LIN {X 0,Y 142.881,Z 390.405,A -85,B 0,C 180,E1 -25256.55,E2 -25256.55} C_VEL
LIN {X 0,Y 141.554,Z 401.416,A -85,B 0,C 180,E1 -25257.538,E2 -25257.538} C_VEL
LIN {X 0,Y 139.699,Z 412.081,A -85,B 0,C 180,E1 -25259.036,E2 -25259.036} C_VEL
LIN {X 0,Y 138.159,Z 420.57,A -85,B 0,C 180,E1 -25260.686,E2 -25260.686} C_VEL
LIN {X 0,Y 135.961,Z 428.897,A -85,B 0,C 180,E1 -25262.694,E2 -25262.694} C_VEL
LIN {X 0,Y 133.997,Z 436.865,A -85,B 0,C 180,E1 -25265.192,E2 -25265.192} C_VEL
LIN {X 0,Y 131.868,Z 444.276,A -85,B 0,C 180,E1 -25268.096,E2 -25268.096} C_VEL
LIN {X 0,Y 129.751,Z 451.798,A -85,B 0,C 180,E1 -25271.854,E2 -25271.854} C_VEL
LIN {X 0,Y 128.143,Z 457.67,A -85,B 0,C 180,E1 -25275.712,E2 -25275.712} C_VEL
LIN {X 0,Y 127.32,Z 461.5,A -85,B 0,C 180,E1 -25278.861,E2 -25278.861} C_VEL
LIN {X 0,Y 126.556,Z 465.852,A -85,B 0,C 180,E1 -25283.623,E2 -25283.623} C_VEL
LIN {X 0,Y 126.391,Z 468.069,A -85,B 0,C 180,E1 -25286.812,E2 -25286.812} C_VEL
LIN {X 0,Y 126.467,Z 469.672,A -85,B 0,C 180,E1 -25290,E2 -25290} C_VEL
LIN {X 0,Y 126.376,Z 470.674,A -85,B 0,C 180,E1 -25293.188,E2 -25293.188} C_VEL
LIN {X 0,Y 126.521,Z 471.21,A -85,B 0,C 180,E1 -25296.378,E2 -25296.378} C_VEL
LIN {X 0,Y 126.968,Z 471.301,A -85,B 0,C 180,E1 -25299.558,E2 -25299.558} C_VEL
LIN {X 0,Y 127.775,Z 470.915,A -85,B 0,C 180,E1 -25302.709,E2 -25302.709} C_VEL
LIN {X 0,Y 128.973,Z 469.949,A -85,B 0,C 180,E1 -25305.81,E2 -25305.81} C_VEL
LIN {X 0,Y 130.517,Z 468.51,A -85,B 0,C 180,E1 -25308.849,E2 -25308.849} C_VEL
LIN {X 0,Y 133.483,Z 465.427,A -85,B 0,C 180,E1 -25313.258,E2 -25313.258} C_VEL
LIN {X 0,Y 137.366,Z 461.085,A -85,B 0,C 180,E1 -25317.416,E2 -25317.416} C_VEL
LIN {X 0,Y 141.882,Z 455.129,A -85,B 0,C 180,E1 -25321.338,E2 -25321.338} C_VEL
LIN {X 0,Y 146.264,Z 448.82,A -85,B 0,C 180,E1 -25324.372,E2 -25324.372} C_VEL
LIN {X 0,Y 149.954,Z 442.696,A -85,B 0,C 180,E1 -25326.694,E2 -25326.694} C_VEL
LIN {X 0,Y 153.372,Z 436.478,A -85,B 0,C 180,E1 -25328.55,E2 -25328.55} C_VEL
LIN {X 0,Y 156.553,Z 429.785,A -85,B 0,C 180,E1 -25330.188,E2 -25330.188} C_VEL
LIN {X 0,Y 159.841,Z 421.95,A -85,B 0,C 180,E1 -25331.683,E2 -25331.683} C_VEL
LIN {X 0,Y 162.735,Z 413.909,A -85,B 0,C 180,E1 -25332.857,E2 -25332.857} C_VEL
LIN {X 0,Y 165.005,Z 406.242,A -85,B 0,C 180,E1 -25333.73,E2 -25333.73} C_VEL
LIN {X 0,Y 165.605,Z 401.983,A -85,B 0,C 180,E1 -25334.367,E2 -25334.367} C_VEL
LIN {X 0,Y 164.474,Z 391.08,A -85,B 0,C 180,E1 -25336.71,E2 -25336.71} C_VEL
LIN {X 0,Y 164.587,Z 387.258,A -85,B 0,C 180,E1 -25337.085,E2 -25337.085} C_VEL
LIN {X 0,Y 165.584,Z 377.046,A -85,B 0,C 180,E1 -25337.548,E2 -25337.548} C_VEL
LIN {X 0,Y 163.149,Z 370.127,A -85,B 0,C 180,E1 -25339.553,E2 -25339.553} C_VEL
LIN {X 0,Y 160.189,Z 363.188,A -85,B 0,C 180,E1 -25342.105,E2 -25342.105} C_VEL
LIN {X 0,Y 157.036,Z 356.535,A -85,B 0,C 180,E1 -25345.217,E2 -25345.217} C_VEL
LIN {X 0,Y 155.41,Z 353.618,A -85,B 0,C 180,E1 -25346.981,E2 -25346.981} C_VEL
LIN {X 0,Y 152.992,Z 349.888,A -85,B 0,C 180,E1 -25349.954,E2 -25349.954} C_VEL
LIN {X 0,Y 150.142,Z 345.841,A -85,B 0,C 180,E1 -25354.422,E2 -25354.422} C_VEL
LIN {X 0,Y 149.876,Z 345.124,A -85,B 0,C 180,E1 -25355.038,E2 -25355.038} C_VEL
LIN {X 0,Y 147.126,Z 341.865,A -85,B 0,C 180,E1 -25364.768,E2 -25364.768} C_VEL
LIN {X 0,Y 147.088,Z 341.6,A -85,B 0,C 180,E1 -25366.178,E2 -25366.178} C_VEL
LIN {X 0,Y 147.398,Z 341.979,A -85,B 0,C 180,E1 -25369.849,E2 -25369.849} C_VEL
LIN {X 0,Y 149.892,Z 344.586,A -85,B 0,C 180,E1 -25377.313,E2 -25377.313} C_VEL
LIN {X 0,Y 150.355,Z 345.232,A -85,B 0,C 180,E1 -25378.236,E2 -25378.236} C_VEL
LIN {X 0,Y 152.17,Z 348.533,A -85,B 0,C 180,E1 -25381.324,E2 -25381.324} C_VEL
LIN {X 0,Y 153.507,Z 350.114,A -85,B 0,C 180,E1 -25383.105,E2 -25383.105} C_VEL
LIN {X 0,Y 156.121,Z 354.377,A -85,B 0,C 180,E1 -25386.209,E2 -25386.209} C_VEL
LIN {X 0,Y 159.1,Z 359.359,A -85,B 0,C 180,E1 -25389.17,E2 -25389.17} C_VEL
LIN {X 0,Y 162.048,Z 364.517,A -85,B 0,C 180,E1 -25391.701,E2 -25391.701} C_VEL
LIN {X 0,Y 165.657,Z 371.579,A -85,B 0,C 180,E1 -25394.47,E2 -25394.47} C_VEL
LIN {X 0,Y 165.925,Z 372.264,A -85,B 0,C 180,E1 -25394.677,E2 -25394.677} C_VEL
LIN {X 0,Y 164.165,Z 387.712,A -85,B 0,C 180,E1 -25395.387,E2 -25395.387} C_VEL
LIN {X 0,Y 162.262,Z 397.3,A -85,B 0,C 180,E1 -25396.153,E2 -25396.153} C_VEL
LIN {X 0,Y 159.595,Z 407.073,A -85,B 0,C 180,E1 -25397.253,E2 -25397.253} C_VEL
LIN {X 0,Y 156.834,Z 415.193,A -85,B 0,C 180,E1 -25398.467,E2 -25398.467} C_VEL
LIN {X 0,Y 153.338,Z 423.473,A -85,B 0,C 180,E1 -25400.023,E2 -25400.023} C_VEL
LIN {X 0,Y 149.693,Z 430.879,A -85,B 0,C 180,E1 -25401.83,E2 -25401.83} C_VEL
LIN {X 0,Y 145.991,Z 437.405,A -85,B 0,C 180,E1 -25403.847,E2 -25403.847} C_VEL
LIN {X 0,Y 141.45,Z 444.337,A -85,B 0,C 180,E1 -25406.581,E2 -25406.581} C_VEL
LIN {X 0,Y 137.261,Z 449.948,A -85,B 0,C 180,E1 -25409.495,E2 -25409.495} C_VEL
LIN {X 0,Y 133.417,Z 454.459,A -85,B 0,C 180,E1 -25412.563,E2 -25412.563} C_VEL
LIN {X 0,Y 129.233,Z 458.881,A -85,B 0,C 180,E1 -25416.742,E2 -25416.742} C_VEL
LIN {X 0,Y 127.087,Z 460.797,A -85,B 0,C 180,E1 -25419.269,E2 -25419.269} C_VEL
LIN {X 0,Y 124.55,Z 462.795,A -85,B 0,C 180,E1 -25422.817,E2 -25422.817} C_VEL
LIN {X 0,Y 121.52,Z 464.62,A -85,B 0,C 180,E1 -25428.751,E2 -25428.751} C_VEL
LIN {X 0,Y 119.539,Z 464.603,A -85,B 0,C 180,E1 -25435.397,E2 -25435.397} C_VEL
LIN {X 0,Y 119.135,Z 464.109,A -85,B 0,C 180,E1 -25437.933,E2 -25437.933} C_VEL
LIN {X 0,Y 118.875,Z 462.498,A -85,B 0,C 180,E1 -25442.476,E2 -25442.476} C_VEL
LIN {X 0,Y 119.08,Z 460.912,A -85,B 0,C 180,E1 -25445.599,E2 -25445.599} C_VEL
LIN {X 0,Y 119.74,Z 457.829,A -85,B 0,C 180,E1 -25449.903,E2 -25449.903} C_VEL
LIN {X 0,Y 121.008,Z 452.9,A -85,B 0,C 180,E1 -25454.85,E2 -25454.85} C_VEL
LIN {X 0,Y 122.587,Z 447.322,A -85,B 0,C 180,E1 -25459.097,E2 -25459.097} C_VEL
LIN {X 0,Y 124.429,Z 441.266,A -85,B 0,C 180,E1 -25462.699,E2 -25462.699} C_VEL
LIN {X 0,Y 126.768,Z 433.558,A -85,B 0,C 180,E1 -25466.309,E2 -25466.309} C_VEL
LIN {X 0,Y 129.417,Z 424.126,A -85,B 0,C 180,E1 -25469.611,E2 -25469.611} C_VEL
LIN {X 0,Y 131.533,Z 415.611,A -85,B 0,C 180,E1 -25471.914,E2 -25471.914} C_VEL
LIN {X 0,Y 133.45,Z 406.731,A -85,B 0,C 180,E1 -25473.773,E2 -25473.773} C_VEL
LIN {X 0,Y 134.912,Z 397.798,A -85,B 0,C 180,E1 -25475.218,E2 -25475.218} C_VEL
LIN {X 0,Y 136.377,Z 386.472,A -85,B 0,C 180,E1 -25476.512,E2 -25476.512} C_VEL
LIN {X 0,Y 137.535,Z 371.795,A -85,B 0,C 180,E1 -25477.412,E2 -25477.412} C_VEL
LIN {X 0,Y 138.736,Z 349.669,A -85,B 0,C 180,E1 -25478.553,E2 -25478.553} C_VEL
LIN {X 0,Y 136.797,Z 343.639,A -85,B 0,C 180,E1 -25479.381,E2 -25479.381} C_VEL
LIN {X 0,Y 128.682,Z 327.088,A -85,B 0,C 180,E1 -25482.589,E2 -25482.589} C_VEL
LIN {X 0,Y 123.725,Z 318.724,A -85,B 0,C 180,E1 -25484.659,E2 -25484.659} C_VEL
LIN {X 0,Y 122.333,Z 316.065,A -85,B 0,C 180,E1 -25485.299,E2 -25485.299} C_VEL
LIN {X 0,Y 122.147,Z 315.082,A -85,B 0,C 180,E1 -25485.541,E2 -25485.541} C_VEL
LIN {X 0,Y 122.023,Z 315.065,A -85,B 0,C 180,E1 -25492.848,E2 -25492.848} C_VEL
LIN {X 0,Y 121.957,Z 315.112,A -85,B 0,C 180,E1 -25497.452,E2 -25497.452} C_VEL
LIN {X 0,Y 121.904,Z 315.107,A -85,B 0,C 180,E1 -25501.255,E2 -25501.255} C_VEL
LIN {X 0,Y 121.886,Z 315.116,A -85,B 0,C 180,E1 -25506.171,E2 -25506.171} C_VEL
LIN {X 0,Y 121.88,Z 315.098,A -85,B 0,C 180,E1 -25511.442,E2 -25511.442} C_VEL
LIN {X 0,Y 121.925,Z 315.109,A -85,B 0,C 180,E1 -25518.532,E2 -25518.532} C_VEL
LIN {X 0,Y 121.95,Z 315.077,A -85,B 0,C 180,E1 -25524.809,E2 -25524.809} C_VEL
LIN {X 0,Y 121.927,Z 315.105,A -85,B 0,C 180,E1 -25529.836,E2 -25529.836} C_VEL
LIN {X 0,Y 121.98,Z 315.086,A -85,B 0,C 180,E1 -25536.214,E2 -25536.214} C_VEL
LIN {X 0,Y 122.04,Z 315.06,A -85,B 0,C 180,E1 -25539.786,E2 -25539.786} C_VEL
LIN {X 0,Y 122.236,Z 315.072,A -85,B 0,C 180,E1 -25546.704,E2 -25546.704} C_VEL
LIN {X 0,Y 122.403,Z 315.044,A -85,B 0,C 180,E1 -25550.081,E2 -25550.081} C_VEL
LIN {X 0,Y 122.589,Z 315,A -85,B 0,C 180,E1 -25556.713,E2 -25556.713} C_VEL
LIN {X 0,Y 123.036,Z 314.966,A -85,B 0,C 180,E1 -25560,E2 -25560} C_VEL
LIN {X 0,Y 122.419,Z 315.034,A -85,B 0,C 180,E1 -25566.593,E2 -25566.593} C_VEL
LIN {X 0,Y 122.319,Z 315.049,A -85,B 0,C 180,E1 -25572.385,E2 -25572.385} C_VEL
LIN {X 0,Y 122.1,Z 315.087,A -85,B 0,C 180,E1 -25576.726,E2 -25576.726} C_VEL
LIN {X 0,Y 122.024,Z 315.084,A -85,B 0,C 180,E1 -25582.855,E2 -25582.855} C_VEL
LIN {X 0,Y 121.937,Z 315.108,A -85,B 0,C 180,E1 -25587.457,E2 -25587.457} C_VEL
LIN {X 0,Y 121.896,Z 315.103,A -85,B 0,C 180,E1 -25591.258,E2 -25591.258} C_VEL
LIN {X 0,Y 121.88,Z 315.114,A -85,B 0,C 180,E1 -25596.171,E2 -25596.171} C_VEL
LIN {X 0,Y 121.861,Z 315.085,A -85,B 0,C 180,E1 -25601.434,E2 -25601.434} C_VEL
LIN {X 0,Y 121.869,Z 315.22,A -85,B 0,C 180,E1 -25606.089,E2 -25606.089} C_VEL
LIN {X 0,Y 122.984,Z 318.162,A -85,B 0,C 180,E1 -25606.67,E2 -25606.67} C_VEL
LIN {X 0,Y 124.377,Z 320.409,A -85,B 0,C 180,E1 -25607.271,E2 -25607.271} C_VEL
LIN {X 0,Y 129.513,Z 329.802,A -85,B 0,C 180,E1 -25609.438,E2 -25609.438} C_VEL
LIN {X 0,Y 134.184,Z 342.151,A -85,B 0,C 180,E1 -25611.496,E2 -25611.496} C_VEL
LIN {X 0,Y 136.431,Z 349.354,A -85,B 0,C 180,E1 -25612.502,E2 -25612.502} C_VEL
LIN {X 0,Y 137.956,Z 367.641,A -85,B 0,C 180,E1 -25614.015,E2 -25614.015} C_VEL
LIN {X 0,Y 136.489,Z 390.702,A -85,B 0,C 180,E1 -25615.297,E2 -25615.297} C_VEL
LIN {X 0,Y 135.015,Z 402.002,A -85,B 0,C 180,E1 -25616.379,E2 -25616.379} C_VEL
LIN {X 0,Y 133.188,Z 411.946,A -85,B 0,C 180,E1 -25617.848,E2 -25617.848} C_VEL
LIN {X 0,Y 131.625,Z 420.222,A -85,B 0,C 180,E1 -25619.521,E2 -25619.521} C_VEL
LIN {X 0,Y 129.328,Z 428.565,A -85,B 0,C 180,E1 -25621.609,E2 -25621.609} C_VEL
LIN {X 0,Y 127.262,Z 436.553,A -85,B 0,C 180,E1 -25624.222,E2 -25624.222} C_VEL
LIN {X 0,Y 125.304,Z 443.124,A -85,B 0,C 180,E1 -25626.883,E2 -25626.883} C_VEL
LIN {X 0,Y 123.38,Z 449.369,A -85,B 0,C 180,E1 -25630.016,E2 -25630.016} C_VEL
LIN {X 0,Y 121.893,Z 454.554,A -85,B 0,C 180,E1 -25633.245,E2 -25633.245} C_VEL
LIN {X 0,Y 120.763,Z 458.86,A -85,B 0,C 180,E1 -25636.539,E2 -25636.539} C_VEL
LIN {X 0,Y 119.968,Z 462.417,A -85,B 0,C 180,E1 -25639.878,E2 -25639.878} C_VEL
LIN {X 0,Y 119.386,Z 466.474,A -85,B 0,C 180,E1 -25644.934,E2 -25644.934} C_VEL
LIN {X 0,Y 119.315,Z 467.602,A -85,B 0,C 180,E1 -25646.623,E2 -25646.623} C_VEL
LIN {X 0,Y 119.39,Z 469.238,A -85,B 0,C 180,E1 -25650,E2 -25650} C_VEL
LIN {X 0,Y 119.285,Z 470.332,A -85,B 0,C 180,E1 -25653.378,E2 -25653.378} C_VEL
LIN {X 0,Y 119.462,Z 470.963,A -85,B 0,C 180,E1 -25656.757,E2 -25656.757} C_VEL
LIN {X 0,Y 119.972,Z 471.15,A -85,B 0,C 180,E1 -25660.121,E2 -25660.121} C_VEL
LIN {X 0,Y 120.85,Z 470.781,A -85,B 0,C 180,E1 -25663.451,E2 -25663.451} C_VEL
LIN {X 0,Y 122.135,Z 469.894,A -85,B 0,C 180,E1 -25666.721,E2 -25666.721} C_VEL
LIN {X 0,Y 123.811,Z 468.554,A -85,B 0,C 180,E1 -25669.912,E2 -25669.912} C_VEL
LIN {X 0,Y 127,Z 465.575,A -85,B 0,C 180,E1 -25674.521,E2 -25674.521} C_VEL
LIN {X 0,Y 129.642,Z 462.894,A -85,B 0,C 180,E1 -25677.437,E2 -25677.437} C_VEL
LIN {X 0,Y 134.245,Z 457.71,A -85,B 0,C 180,E1 -25681.567,E2 -25681.567} C_VEL
LIN {X 0,Y 138.626,Z 452.168,A -85,B 0,C 180,E1 -25684.773,E2 -25684.773} C_VEL
LIN {X 0,Y 143.403,Z 445.255,A -85,B 0,C 180,E1 -25687.777,E2 -25687.777} C_VEL
LIN {X 0,Y 147.966,Z 437.517,A -85,B 0,C 180,E1 -25690.27,E2 -25690.27} C_VEL
LIN {X 0,Y 152.028,Z 429.463,A -85,B 0,C 180,E1 -25692.268,E2 -25692.268} C_VEL
LIN {X 0,Y 155.268,Z 422.18,A -85,B 0,C 180,E1 -25693.65,E2 -25693.65} C_VEL
LIN {X 0,Y 158.274,Z 414.242,A -85,B 0,C 180,E1 -25694.821,E2 -25694.821} C_VEL
LIN {X 0,Y 160.984,Z 405.406,A -85,B 0,C 180,E1 -25695.812,E2 -25695.812} C_VEL
LIN {X 0,Y 163.083,Z 396.249,A -85,B 0,C 180,E1 -25696.588,E2 -25696.588} C_VEL
LIN {X 0,Y 164.587,Z 387.258,A -85,B 0,C 180,E1 -25697.085,E2 -25697.085} C_VEL
LIN {X 0,Y 164.625,Z 384.216,A -85,B 0,C 180,E1 -25697.418,E2 -25697.418} C_VEL
LIN {X 0,Y 163.648,Z 380.573,A -85,B 0,C 180,E1 -25698.321,E2 -25698.321} C_VEL
LIN {X 0,Y 162.806,Z 378.841,A -85,B 0,C 180,E1 -25698.965,E2 -25698.965} C_VEL
LIN {X 0,Y 158.938,Z 372.15,A -85,B 0,C 180,E1 -25702.014,E2 -25702.014} C_VEL
LIN {X 0,Y 156.045,Z 365.237,A -85,B 0,C 180,E1 -25704.964,E2 -25704.964} C_VEL
LIN {X 0,Y 153.632,Z 360.182,A -85,B 0,C 180,E1 -25707.728,E2 -25707.728} C_VEL
LIN {X 0,Y 151.299,Z 356.419,A -85,B 0,C 180,E1 -25710.824,E2 -25710.824} C_VEL
LIN {X 0,Y 148.68,Z 352.346,A -85,B 0,C 180,E1 -25715.359,E2 -25715.359} C_VEL
LIN {X 0,Y 148.117,Z 351.687,A -85,B 0,C 180,E1 -25716.594,E2 -25716.594} C_VEL
LIN {X 0,Y 146.134,Z 348.78,A -85,B 0,C 180,E1 -25725.376,E2 -25725.376} C_VEL
LIN {X 0,Y 146.36,Z 348.904,A -85,B 0,C 180,E1 -25729.355,E2 -25729.355} C_VEL
LIN {X 0,Y 148.716,Z 351.517,A -85,B 0,C 180,E1 -25736.953,E2 -25736.953} C_VEL
LIN {X 0,Y 150.98,Z 355.613,A -85,B 0,C 180,E1 -25741.112,E2 -25741.112} C_VEL
LIN {X 0,Y 151.99,Z 357.05,A -85,B 0,C 180,E1 -25742.54,E2 -25742.54} C_VEL
LIN {X 0,Y 154.147,Z 360.784,A -85,B 0,C 180,E1 -25745.304,E2 -25745.304} C_VEL
LIN {X 0,Y 157.613,Z 366.789,A -85,B 0,C 180,E1 -25748.904,E2 -25748.904} C_VEL
LIN {X 0,Y 161.88,Z 375.319,A -85,B 0,C 180,E1 -25752.643,E2 -25752.643} C_VEL
LIN {X 0,Y 160.367,Z 387.956,A -85,B 0,C 180,E1 -25753.275,E2 -25753.275} C_VEL
LIN {X 0,Y 158.275,Z 397.956,A -85,B 0,C 180,E1 -25754.078,E2 -25754.078} C_VEL
LIN {X 0,Y 155.458,Z 407.697,A -85,B 0,C 180,E1 -25755.17,E2 -25755.17} C_VEL
LIN {X 0,Y 152.131,Z 416.773,A -85,B 0,C 180,E1 -25756.553,E2 -25756.553} C_VEL
LIN {X 0,Y 148.716,Z 424.307,A -85,B 0,C 180,E1 -25758.005,E2 -25758.005} C_VEL
LIN {X 0,Y 144.809,Z 431.748,A -85,B 0,C 180,E1 -25759.861,E2 -25759.861} C_VEL
LIN {X 0,Y 140.404,Z 438.966,A -85,B 0,C 180,E1 -25762.181,E2 -25762.181} C_VEL
LIN {X 0,Y 134.426,Z 447.162,A -85,B 0,C 180,E1 -25765.739,E2 -25765.739} C_VEL
LIN {X 0,Y 131.257,Z 451.035,A -85,B 0,C 180,E1 -25767.943,E2 -25767.943} C_VEL
LIN {X 0,Y 127.214,Z 455.365,A -85,B 0,C 180,E1 -25771.099,E2 -25771.099} C_VEL
LIN {X 0,Y 123.456,Z 458.98,A -85,B 0,C 180,E1 -25774.7,E2 -25774.7} C_VEL
LIN {X 0,Y 120.51,Z 461.436,A -85,B 0,C 180,E1 -25778.068,E2 -25778.068} C_VEL
LIN {X 0,Y 116.677,Z 463.957,A -85,B 0,C 180,E1 -25783.714,E2 -25783.714} C_VEL
LIN {X 0,Y 114.749,Z 464.846,A -85,B 0,C 180,E1 -25787.647,E2 -25787.647} C_VEL
LIN {X 0,Y 113.333,Z 465.087,A -85,B 0,C 180,E1 -25791.677,E2 -25791.677} C_VEL
LIN {X 0,Y 112.367,Z 464.659,A -85,B 0,C 180,E1 -25795.744,E2 -25795.744} C_VEL
LIN {X 0,Y 111.773,Z 462.831,A -85,B 0,C 180,E1 -25801.677,E2 -25801.677} C_VEL
LIN {X 0,Y 112.31,Z 459.382,A -85,B 0,C 180,E1 -25807.948,E2 -25807.948} C_VEL
LIN {X 0,Y 113.072,Z 456.268,A -85,B 0,C 180,E1 -25811.895,E2 -25811.895} C_VEL
LIN {X 0,Y 114.125,Z 452.411,A -85,B 0,C 180,E1 -25815.74,E2 -25815.74} C_VEL
LIN {X 0,Y 115.945,Z 446.423,A -85,B 0,C 180,E1 -25820.405,E2 -25820.405} C_VEL
LIN {X 0,Y 118.369,Z 438.758,A -85,B 0,C 180,E1 -25824.891,E2 -25824.891} C_VEL
LIN {X 0,Y 120.764,Z 430.977,A -85,B 0,C 180,E1 -25828.333,E2 -25828.333} C_VEL
LIN {X 0,Y 122.829,Z 423.921,A -85,B 0,C 180,E1 -25830.82,E2 -25830.82} C_VEL
LIN {X 0,Y 125.081,Z 415.306,A -85,B 0,C 180,E1 -25833.221,E2 -25833.221} C_VEL
LIN {X 0,Y 127.001,Z 406.766,A -85,B 0,C 180,E1 -25835.065,E2 -25835.065} C_VEL
LIN {X 0,Y 128.531,Z 397.81,A -85,B 0,C 180,E1 -25836.565,E2 -25836.565} C_VEL
LIN {X 0,Y 130.127,Z 385.909,A -85,B 0,C 180,E1 -25837.948,E2 -25837.948} C_VEL
LIN {X 0,Y 131.444,Z 369.026,A -85,B 0,C 180,E1 -25838.966,E2 -25838.966} C_VEL
LIN {X 0,Y 132.421,Z 350.923,A -85,B 0,C 180,E1 -25839.948,E2 -25839.948} C_VEL
LIN {X 0,Y 131.134,Z 347.005,A -85,B 0,C 180,E1 -25840.537,E2 -25840.537} C_VEL
LIN {X 0,Y 123.12,Z 330.389,A -85,B 0,C 180,E1 -25843.974,E2 -25843.974} C_VEL
LIN {X 0,Y 116.777,Z 319.818,A -85,B 0,C 180,E1 -25846.876,E2 -25846.876} C_VEL
LIN {X 0,Y 115.222,Z 317.086,A -85,B 0,C 180,E1 -25847.666,E2 -25847.666} C_VEL
LIN {X 0,Y 114.975,Z 315.967,A -85,B 0,C 180,E1 -25847.911,E2 -25847.911} C_VEL
LIN {X 0,Y 114.946,Z 315.95,A -85,B 0,C 180,E1 -25853.49,E2 -25853.49} C_VEL
LIN {X 0,Y 114.862,Z 315.984,A -85,B 0,C 180,E1 -25861.061,E2 -25861.061} C_VEL
LIN {X 0,Y 114.782,Z 316.001,A -85,B 0,C 180,E1 -25867.754,E2 -25867.754} C_VEL
LIN {X 0,Y 114.807,Z 315.975,A -85,B 0,C 180,E1 -25872.727,E2 -25872.727} C_VEL
LIN {X 0,Y 114.844,Z 315.992,A -85,B 0,C 180,E1 -25877.688,E2 -25877.688} C_VEL
LIN {X 0,Y 114.847,Z 315.971,A -85,B 0,C 180,E1 -25882.703,E2 -25882.703} C_VEL
LIN {X 0,Y 114.862,Z 315.983,A -85,B 0,C 180,E1 -25888.935,E2 -25888.935} C_VEL
LIN {X 0,Y 114.945,Z 315.96,A -85,B 0,C 180,E1 -25896.507,E2 -25896.507} C_VEL
LIN {X 0,Y 115.007,Z 315.953,A -85,B 0,C 180,E1 -25902.209,E2 -25902.209} C_VEL
LIN {X 0,Y 115.252,Z 315.941,A -85,B 0,C 180,E1 -25907.327,E2 -25907.327} C_VEL
LIN {X 0,Y 115.359,Z 315.901,A -85,B 0,C 180,E1 -25913.001,E2 -25913.001} C_VEL
LIN {X 0,Y 115.988,Z 315.844,A -85,B 0,C 180,E1 -25920,E2 -25920} C_VEL
LIN {X 0,Y 115.36,Z 315.909,A -85,B 0,C 180,E1 -25926.998,E2 -25926.998} C_VEL
LIN {X 0,Y 115.252,Z 315.931,A -85,B 0,C 180,E1 -25932.671,E2 -25932.671} C_VEL
LIN {X 0,Y 115.004,Z 315.967,A -85,B 0,C 180,E1 -25937.791,E2 -25937.791} C_VEL
LIN {X 0,Y 114.944,Z 315.97,A -85,B 0,C 180,E1 -25943.492,E2 -25943.492} C_VEL
LIN {X 0,Y 114.853,Z 315.979,A -85,B 0,C 180,E1 -25951.057,E2 -25951.057} C_VEL
LIN {X 0,Y 114.774,Z 315.986,A -85,B 0,C 180,E1 -25957.758,E2 -25957.758} C_VEL
LIN {X 0,Y 114.784,Z 315.984,A -85,B 0,C 180,E1 -25963.678,E2 -25963.678} C_VEL
LIN {X 0,Y 115.813,Z 318.882,A -85,B 0,C 180,E1 -25964.3,E2 -25964.3} C_VEL
LIN {X 0,Y 117.212,Z 320.888,A -85,B 0,C 180,E1 -25964.962,E2 -25964.962} C_VEL
LIN {X 0,Y 123.967,Z 333.026,A -85,B 0,C 180,E1 -25968.08,E2 -25968.08} C_VEL
LIN {X 0,Y 128.513,Z 345.387,A -85,B 0,C 180,E1 -25970.267,E2 -25970.267} C_VEL
LIN {X 0,Y 130.313,Z 351.13,A -85,B 0,C 180,E1 -25971.138,E2 -25971.138} C_VEL
LIN {X 0,Y 131.654,Z 368.464,A -85,B 0,C 180,E1 -25972.646,E2 -25972.646} C_VEL
LIN {X 0,Y 130.172,Z 390.427,A -85,B 0,C 180,E1 -25973.916,E2 -25973.916} C_VEL
LIN {X 0,Y 128.515,Z 402.447,A -85,B 0,C 180,E1 -25975.131,E2 -25975.131} C_VEL
LIN {X 0,Y 126.537,Z 412.644,A -85,B 0,C 180,E1 -25976.739,E2 -25976.739} C_VEL
LIN {X 0,Y 124.736,Z 421.206,A -85,B 0,C 180,E1 -25978.59,E2 -25978.59} C_VEL
LIN {X 0,Y 122.381,Z 429.343,A -85,B 0,C 180,E1 -25980.783,E2 -25980.783} C_VEL
LIN {X 0,Y 120.568,Z 436.148,A -85,B 0,C 180,E1 -25983.145,E2 -25983.145} C_VEL
LIN {X 0,Y 118.219,Z 443.608,A -85,B 0,C 180,E1 -25986.342,E2 -25986.342} C_VEL
LIN {X 0,Y 115.874,Z 451.178,A -85,B 0,C 180,E1 -25990.514,E2 -25990.514} C_VEL
LIN {X 0,Y 113.861,Z 458.084,A -85,B 0,C 180,E1 -25995.706,E2 -25995.706} C_VEL
LIN {X 0,Y 112.682,Z 463.288,A -85,B 0,C 180,E1 -26001.03,E2 -26001.03} C_VEL
LIN {X 0,Y 112.245,Z 467.079,A -85,B 0,C 180,E1 -26006.41,E2 -26006.41} C_VEL
LIN {X 0,Y 112.301,Z 468.797,A -85,B 0,C 180,E1 -26010,E2 -26010} C_VEL
LIN {X 0,Y 112.204,Z 469.989,A -85,B 0,C 180,E1 -26013.591,E2 -26013.591} C_VEL
LIN {X 0,Y 112.425,Z 470.718,A -85,B 0,C 180,E1 -26017.182,E2 -26017.182} C_VEL
LIN {X 0,Y 112.973,Z 470.964,A -85,B 0,C 180,E1 -26020.756,E2 -26020.756} C_VEL
LIN {X 0,Y 113.955,Z 470.632,A -85,B 0,C 180,E1 -26024.281,E2 -26024.281} C_VEL
LIN {X 0,Y 115.335,Z 469.846,A -85,B 0,C 180,E1 -26027.738,E2 -26027.738} C_VEL
LIN {X 0,Y 117.137,Z 468.613,A -85,B 0,C 180,E1 -26031.099,E2 -26031.099} C_VEL
LIN {X 0,Y 119.277,Z 466.907,A -85,B 0,C 180,E1 -26034.358,E2 -26034.358} C_VEL
LIN {X 0,Y 123.4,Z 463.19,A -85,B 0,C 180,E1 -26038.952,E2 -26038.952} C_VEL
LIN {X 0,Y 126.608,Z 460.041,A -85,B 0,C 180,E1 -26041.825,E2 -26041.825} C_VEL
LIN {X 0,Y 130.964,Z 455.07,A -85,B 0,C 180,E1 -26045.23,E2 -26045.23} C_VEL
LIN {X 0,Y 135.807,Z 448.852,A -85,B 0,C 180,E1 -26048.388,E2 -26048.388} C_VEL
LIN {X 0,Y 139.922,Z 442.814,A -85,B 0,C 180,E1 -26050.764,E2 -26050.764} C_VEL
LIN {X 0,Y 144.471,Z 435.495,A -85,B 0,C 180,E1 -26052.924,E2 -26052.924} C_VEL
LIN {X 0,Y 148.499,Z 427.674,A -85,B 0,C 180,E1 -26054.773,E2 -26054.773} C_VEL
LIN {X 0,Y 152.778,Z 418.092,A -85,B 0,C 180,E1 -26056.427,E2 -26056.427} C_VEL
LIN {X 0,Y 156.539,Z 407.168,A -85,B 0,C 180,E1 -26057.775,E2 -26057.775} C_VEL
LIN {X 0,Y 159.103,Z 396.879,A -85,B 0,C 180,E1 -26058.669,E2 -26058.669} C_VEL
LIN {X 0,Y 160.801,Z 387.378,A -85,B 0,C 180,E1 -26059.194,E2 -26059.194} C_VEL
LIN {X 0,Y 161.595,Z 379.591,A -85,B 0,C 180,E1 -26059.586,E2 -26059.586} C_VEL
LIN {X 0,Y 158.938,Z 372.15,A -85,B 0,C 180,E1 -26062.014,E2 -26062.014} C_VEL
LIN {X 0,Y 157.126,Z 368.923,A -85,B 0,C 180,E1 -26063.678,E2 -26063.678} C_VEL
LIN {X 0,Y 155.073,Z 366.798,A -85,B 0,C 180,E1 -26065.573,E2 -26065.573} C_VEL
LIN {X 0,Y 149.985,Z 363.317,A -85,B 0,C 180,E1 -26071.22,E2 -26071.22} C_VEL
LIN {X 0,Y 149.019,Z 362.194,A -85,B 0,C 180,E1 -26072.677,E2 -26072.677} C_VEL
LIN {X 0,Y 147.203,Z 358.783,A -85,B 0,C 180,E1 -26076.44,E2 -26076.44} C_VEL
LIN {X 0,Y 145.162,Z 355.8,A -85,B 0,C 180,E1 -26085.527,E2 -26085.527} C_VEL
LIN {X 0,Y 145.378,Z 355.962,A -85,B 0,C 180,E1 -26089.282,E2 -26089.282} C_VEL
LIN {X 0,Y 147.565,Z 358.67,A -85,B 0,C 180,E1 -26096.681,E2 -26096.681} C_VEL
LIN {X 0,Y 149.493,Z 362.333,A -85,B 0,C 180,E1 -26100.45,E2 -26100.45} C_VEL
LIN {X 0,Y 150.444,Z 363.88,A -85,B 0,C 180,E1 -26101.897,E2 -26101.897} C_VEL
LIN {X 0,Y 152.206,Z 367.144,A -85,B 0,C 180,E1 -26104.334,E2 -26104.334} C_VEL
LIN {X 0,Y 155.341,Z 372.917,A -85,B 0,C 180,E1 -26107.862,E2 -26107.862} C_VEL
LIN {X 0,Y 158.062,Z 378.69,A -85,B 0,C 180,E1 -26110.547,E2 -26110.547} C_VEL
LIN {X 0,Y 157.092,Z 386.489,A -85,B 0,C 180,E1 -26110.967,E2 -26110.967} C_VEL
LIN {X 0,Y 154.613,Z 398.16,A -85,B 0,C 180,E1 -26111.842,E2 -26111.842} C_VEL
LIN {X 0,Y 151.465,Z 408.522,A -85,B 0,C 180,E1 -26112.999,E2 -26112.999} C_VEL
LIN {X 0,Y 148.283,Z 416.813,A -85,B 0,C 180,E1 -26114.259,E2 -26114.259} C_VEL
LIN {X 0,Y 144.31,Z 425.165,A -85,B 0,C 180,E1 -26115.857,E2 -26115.857} C_VEL
LIN {X 0,Y 139.511,Z 433.719,A -85,B 0,C 180,E1 -26118.045,E2 -26118.045} C_VEL
LIN {X 0,Y 134.143,Z 441.613,A -85,B 0,C 180,E1 -26120.797,E2 -26120.797} C_VEL
LIN {X 0,Y 128.779,Z 448.23,A -85,B 0,C 180,E1 -26123.924,E2 -26123.924} C_VEL
LIN {X 0,Y 124.494,Z 452.883,A -85,B 0,C 180,E1 -26126.848,E2 -26126.848} C_VEL
LIN {X 0,Y 119.325,Z 457.776,A -85,B 0,C 180,E1 -26131.092,E2 -26131.092} C_VEL
LIN {X 0,Y 115.605,Z 460.789,A -85,B 0,C 180,E1 -26134.847,E2 -26134.847} C_VEL
LIN {X 0,Y 112.478,Z 462.921,A -85,B 0,C 180,E1 -26138.67,E2 -26138.67} C_VEL
LIN {X 0,Y 111.133,Z 463.79,A -85,B 0,C 180,E1 -26140.637,E2 -26140.637} C_VEL
LIN {X 0,Y 108.46,Z 464.996,A -85,B 0,C 180,E1 -26145.462,E2 -26145.462} C_VEL
LIN {X 0,Y 107.007,Z 465.263,A -85,B 0,C 180,E1 -26148.947,E2 -26148.947} C_VEL
LIN {X 0,Y 105.747,Z 465.016,A -85,B 0,C 180,E1 -26153.264,E2 -26153.264} C_VEL
LIN {X 0,Y 104.956,Z 464.141,A -85,B 0,C 180,E1 -26157.61,E2 -26157.61} C_VEL
LIN {X 0,Y 104.756,Z 461.695,A -85,B 0,C 180,E1 -26164.147,E2 -26164.147} C_VEL
LIN {X 0,Y 105.365,Z 458.783,A -85,B 0,C 180,E1 -26169.04,E2 -26169.04} C_VEL
LIN {X 0,Y 106.623,Z 454.026,A -85,B 0,C 180,E1 -26174.713,E2 -26174.713} C_VEL
LIN {X 0,Y 107.939,Z 449.638,A -85,B 0,C 180,E1 -26178.736,E2 -26178.736} C_VEL
LIN {X 0,Y 109.732,Z 444.273,A -85,B 0,C 180,E1 -26182.641,E2 -26182.641} C_VEL
LIN {X 0,Y 111.891,Z 437.746,A -85,B 0,C 180,E1 -26186.399,E2 -26186.399} C_VEL
LIN {X 0,Y 113.896,Z 431.606,A -85,B 0,C 180,E1 -26189.248,E2 -26189.248} C_VEL
LIN {X 0,Y 116.33,Z 423.701,A -85,B 0,C 180,E1 -26192.164,E2 -26192.164} C_VEL
LIN {X 0,Y 118.578,Z 415.487,A -85,B 0,C 180,E1 -26194.545,E2 -26194.545} C_VEL
LIN {X 0,Y 120.48,Z 407.495,A -85,B 0,C 180,E1 -26196.355,E2 -26196.355} C_VEL
LIN {X 0,Y 122.207,Z 397.919,A -85,B 0,C 180,E1 -26198.039,E2 -26198.039} C_VEL
LIN {X 0,Y 123.861,Z 386.252,A -85,B 0,C 180,E1 -26199.445,E2 -26199.445} C_VEL
LIN {X 0,Y 125.207,Z 369.939,A -85,B 0,C 180,E1 -26200.472,E2 -26200.472} C_VEL
LIN {X 0,Y 126.353,Z 352.954,A -85,B 0,C 180,E1 -26201.382,E2 -26201.382} C_VEL
LIN {X 0,Y 125.255,Z 349.718,A -85,B 0,C 180,E1 -26201.922,E2 -26201.922} C_VEL
LIN {X 0,Y 117.658,Z 333.85,A -85,B 0,C 180,E1 -26205.435,E2 -26205.435} C_VEL
LIN {X 0,Y 111.759,Z 324.045,A -85,B 0,C 180,E1 -26208.384,E2 -26208.384} C_VEL
LIN {X 0,Y 109.837,Z 320.838,A -85,B 0,C 180,E1 -26209.426,E2 -26209.426} C_VEL
LIN {X 0,Y 108.327,Z 318.481,A -85,B 0,C 180,E1 -26210.257,E2 -26210.257} C_VEL
LIN {X 0,Y 107.936,Z 316.816,A -85,B 0,C 180,E1 -26210.609,E2 -26210.609} C_VEL
LIN {X 0,Y 107.858,Z 316.838,A -85,B 0,C 180,E1 -26214.183,E2 -26214.183} C_VEL
LIN {X 0,Y 107.785,Z 316.86,A -85,B 0,C 180,E1 -26222.042,E2 -26222.042} C_VEL
LIN {X 0,Y 107.694,Z 316.883,A -85,B 0,C 180,E1 -26228.453,E2 -26228.453} C_VEL
LIN {X 0,Y 107.713,Z 316.874,A -85,B 0,C 180,E1 -26235.865,E2 -26235.865} C_VEL
LIN {X 0,Y 107.745,Z 316.864,A -85,B 0,C 180,E1 -26241.51,E2 -26241.51} C_VEL
LIN {X 0,Y 107.802,Z 316.858,A -85,B 0,C 180,E1 -26248.563,E2 -26248.563} C_VEL
LIN {X 0,Y 107.909,Z 316.829,A -85,B 0,C 180,E1 -26256.997,E2 -26256.997} C_VEL
LIN {X 0,Y 108.027,Z 316.836,A -85,B 0,C 180,E1 -26264.916,E2 -26264.916} C_VEL
LIN {X 0,Y 108.252,Z 316.81,A -85,B 0,C 180,E1 -26268.768,E2 -26268.768} C_VEL
LIN {X 0,Y 108.437,Z 316.756,A -85,B 0,C 180,E1 -26276.284,E2 -26276.284} C_VEL
LIN {X 0,Y 108.937,Z 316.721,A -85,B 0,C 180,E1 -26280,E2 -26280} C_VEL
LIN {X 0,Y 108.299,Z 316.785,A -85,B 0,C 180,E1 -26287.457,E2 -26287.457} C_VEL
LIN {X 0,Y 108.172,Z 316.814,A -85,B 0,C 180,E1 -26292.959,E2 -26292.959} C_VEL
LIN {X 0,Y 107.898,Z 316.845,A -85,B 0,C 180,E1 -26299.006,E2 -26299.006} C_VEL
LIN {X 0,Y 107.853,Z 316.856,A -85,B 0,C 180,E1 -26304.181,E2 -26304.181} C_VEL
LIN {X 0,Y 107.777,Z 316.864,A -85,B 0,C 180,E1 -26312.039,E2 -26312.039} C_VEL
LIN {X 0,Y 107.681,Z 316.86,A -85,B 0,C 180,E1 -26318.447,E2 -26318.447} C_VEL
LIN {X 0,Y 107.682,Z 317.036,A -85,B 0,C 180,E1 -26320.935,E2 -26320.935} C_VEL
LIN {X 0,Y 108.717,Z 319.741,A -85,B 0,C 180,E1 -26321.618,E2 -26321.618} C_VEL
LIN {X 0,Y 110.366,Z 322.005,A -85,B 0,C 180,E1 -26322.487,E2 -26322.487} C_VEL
LIN {X 0,Y 116.734,Z 333.094,A -85,B 0,C 180,E1 -26325.792,E2 -26325.792} C_VEL
LIN {X 0,Y 119.182,Z 338.199,A -85,B 0,C 180,E1 -26327.003,E2 -26327.003} C_VEL
LIN {X 0,Y 124.112,Z 352.226,A -85,B 0,C 180,E1 -26329.544,E2 -26329.544} C_VEL
LIN {X 0,Y 125.455,Z 368.786,A -85,B 0,C 180,E1 -26331.116,E2 -26331.116} C_VEL
LIN {X 0,Y 123.926,Z 390.084,A -85,B 0,C 180,E1 -26332.388,E2 -26332.388} C_VEL
LIN {X 0,Y 122.323,Z 401.695,A -85,B 0,C 180,E1 -26333.583,E2 -26333.583} C_VEL
LIN {X 0,Y 120.207,Z 412.064,A -85,B 0,C 180,E1 -26335.248,E2 -26335.248} C_VEL
LIN {X 0,Y 118.315,Z 420.705,A -85,B 0,C 180,E1 -26337.179,E2 -26337.179} C_VEL
LIN {X 0,Y 115.845,Z 428.895,A -85,B 0,C 180,E1 -26339.464,E2 -26339.464} C_VEL
LIN {X 0,Y 113.922,Z 435.742,A -85,B 0,C 180,E1 -26341.941,E2 -26341.941} C_VEL
LIN {X 0,Y 111.745,Z 442.382,A -85,B 0,C 180,E1 -26344.88,E2 -26344.88} C_VEL
LIN {X 0,Y 109.616,Z 448.686,A -85,B 0,C 180,E1 -26348.368,E2 -26348.368} C_VEL
LIN {X 0,Y 107.971,Z 453.925,A -85,B 0,C 180,E1 -26351.99,E2 -26351.99} C_VEL
LIN {X 0,Y 106.954,Z 457.306,A -85,B 0,C 180,E1 -26354.762,E2 -26354.762} C_VEL
LIN {X 0,Y 106.013,Z 461.098,A -85,B 0,C 180,E1 -26358.529,E2 -26358.529} C_VEL
LIN {X 0,Y 105.238,Z 465.384,A -85,B 0,C 180,E1 -26364.251,E2 -26364.251} C_VEL
LIN {X 0,Y 105.219,Z 468.352,A -85,B 0,C 180,E1 -26370,E2 -26370} C_VEL
LIN {X 0,Y 105.117,Z 469.64,A -85,B 0,C 180,E1 -26373.833,E2 -26373.833} C_VEL
LIN {X 0,Y 105.369,Z 470.466,A -85,B 0,C 180,E1 -26377.666,E2 -26377.666} C_VEL
LIN {X 0,Y 106.003,Z 470.731,A -85,B 0,C 180,E1 -26381.472,E2 -26381.472} C_VEL
LIN {X 0,Y 107.093,Z 470.486,A -85,B 0,C 180,E1 -26385.218,E2 -26385.218} C_VEL
LIN {X 0,Y 108.583,Z 469.806,A -85,B 0,C 180,E1 -26388.882,E2 -26388.882} C_VEL
LIN {X 0,Y 110.521,Z 468.68,A -85,B 0,C 180,E1 -26392.428,E2 -26392.428} C_VEL
LIN {X 0,Y 114.212,Z 465.931,A -85,B 0,C 180,E1 -26397.484,E2 -26397.484} C_VEL
LIN {X 0,Y 118.885,Z 461.963,A -85,B 0,C 180,E1 -26402.142,E2 -26402.142} C_VEL
LIN {X 0,Y 122.424,Z 458.569,A -85,B 0,C 180,E1 -26405.033,E2 -26405.033} C_VEL
LIN {X 0,Y 126.245,Z 454.497,A -85,B 0,C 180,E1 -26407.759,E2 -26407.759} C_VEL
LIN {X 0,Y 130.35,Z 449.631,A -85,B 0,C 180,E1 -26410.314,E2 -26410.314} C_VEL
LIN {X 0,Y 134.683,Z 443.806,A -85,B 0,C 180,E1 -26412.714,E2 -26412.714} C_VEL
LIN {X 0,Y 139.417,Z 436.719,A -85,B 0,C 180,E1 -26414.887,E2 -26414.887} C_VEL
LIN {X 0,Y 143.595,Z 429.192,A -85,B 0,C 180,E1 -26416.747,E2 -26416.747} C_VEL
LIN {X 0,Y 147.374,Z 421.443,A -85,B 0,C 180,E1 -26418.168,E2 -26418.168} C_VEL
LIN {X 0,Y 150.512,Z 413.805,A -85,B 0,C 180,E1 -26419.254,E2 -26419.254} C_VEL
LIN {X 0,Y 153.521,Z 404.733,A -85,B 0,C 180,E1 -26420.226,E2 -26420.226} C_VEL
LIN {X 0,Y 155.87,Z 395.116,A -85,B 0,C 180,E1 -26421.006,E2 -26421.006} C_VEL
LIN {X 0,Y 157.623,Z 384.723,A -85,B 0,C 180,E1 -26421.533,E2 -26421.533} C_VEL
LIN {X 0,Y 157.822,Z 382.289,A -85,B 0,C 180,E1 -26421.709,E2 -26421.709} C_VEL
LIN {X 0,Y 155.377,Z 375.239,A -85,B 0,C 180,E1 -26424.295,E2 -26424.295} C_VEL
LIN {X 0,Y 152.706,Z 368.676,A -85,B 0,C 180,E1 -26427.423,E2 -26427.423} C_VEL
LIN {X 0,Y 151.427,Z 366.181,A -85,B 0,C 180,E1 -26429.084,E2 -26429.084} C_VEL
LIN {X 0,Y 149.34,Z 362.603,A -85,B 0,C 180,E1 -26432.169,E2 -26432.169} C_VEL
LIN {X 0,Y 149.019,Z 362.194,A -85,B 0,C 180,E1 -26432.677,E2 -26432.677} C_VEL
LIN {X 0,Y 147.738,Z 361.13,A -85,B 0,C 180,E1 -26434.857,E2 -26434.857} C_VEL
LIN {X 0,Y 146.525,Z 361.261,A -85,B 0,C 180,E1 -26437.122,E2 -26437.122} C_VEL
LIN {X 0,Y 144.369,Z 363.119,A -85,B 0,C 180,E1 -26443.365,E2 -26443.365} C_VEL
LIN {X 0,Y 144.21,Z 362.991,A -85,B 0,C 180,E1 -26444.959,E2 -26444.959} C_VEL
LIN {X 0,Y 144.352,Z 362.885,A -85,B 0,C 180,E1 -26448.77,E2 -26448.77} C_VEL
LIN {X 0,Y 146.309,Z 365.64,A -85,B 0,C 180,E1 -26456.147,E2 -26456.147} C_VEL
LIN {X 0,Y 148.713,Z 370.26,A -85,B 0,C 180,E1 -26460.903,E2 -26460.903} C_VEL
LIN {X 0,Y 150.317,Z 373.421,A -85,B 0,C 180,E1 -26463.312,E2 -26463.312} C_VEL
LIN {X 0,Y 153.126,Z 379.085,A -85,B 0,C 180,E1 -26466.799,E2 -26466.799} C_VEL
LIN {X 0,Y 154.476,Z 382.327,A -85,B 0,C 180,E1 -26468.421,E2 -26468.421} C_VEL
LIN {X 0,Y 152.765,Z 392.124,A -85,B 0,C 180,E1 -26468.99,E2 -26468.99} C_VEL
LIN {X 0,Y 150.308,Z 401.728,A -85,B 0,C 180,E1 -26469.815,E2 -26469.815} C_VEL
LIN {X 0,Y 146.91,Z 411.757,A -85,B 0,C 180,E1 -26471.032,E2 -26471.032} C_VEL
LIN {X 0,Y 142.299,Z 421.99,A -85,B 0,C 180,E1 -26472.736,E2 -26472.736} C_VEL
LIN {X 0,Y 137.919,Z 429.876,A -85,B 0,C 180,E1 -26474.496,E2 -26474.496} C_VEL
LIN {X 0,Y 133.69,Z 436.439,A -85,B 0,C 180,E1 -26476.39,E2 -26476.39} C_VEL
LIN {X 0,Y 128.706,Z 443.094,A -85,B 0,C 180,E1 -26478.869,E2 -26478.869} C_VEL
LIN {X 0,Y 124.423,Z 448.089,A -85,B 0,C 180,E1 -26481.257,E2 -26481.257} C_VEL
LIN {X 0,Y 119.729,Z 452.906,A -85,B 0,C 180,E1 -26484.262,E2 -26484.262} C_VEL
LIN {X 0,Y 115.093,Z 457.026,A -85,B 0,C 180,E1 -26487.7,E2 -26487.7} C_VEL
LIN {X 0,Y 110.85,Z 460.337,A -85,B 0,C 180,E1 -26491.594,E2 -26491.594} C_VEL
LIN {X 0,Y 105.946,Z 463.44,A -85,B 0,C 180,E1 -26497.25,E2 -26497.25} C_VEL
LIN {X 0,Y 102.102,Z 465.178,A -85,B 0,C 180,E1 -26503.499,E2 -26503.499} C_VEL
LIN {X 0,Y 99.075,Z 465.282,A -85,B 0,C 180,E1 -26511.288,E2 -26511.288} C_VEL
LIN {X 0,Y 98.205,Z 464.722,A -85,B 0,C 180,E1 -26515.076,E2 -26515.076} C_VEL
LIN {X 0,Y 97.653,Z 463.451,A -85,B 0,C 180,E1 -26519.751,E2 -26519.751} C_VEL
LIN {X 0,Y 97.697,Z 461.517,A -85,B 0,C 180,E1 -26524.431,E2 -26524.431} C_VEL
LIN {X 0,Y 98.254,Z 458.877,A -85,B 0,C 180,E1 -26529.045,E2 -26529.045} C_VEL
LIN {X 0,Y 99.423,Z 454.543,A -85,B 0,C 180,E1 -26534.629,E2 -26534.629} C_VEL
LIN {X 0,Y 101.173,Z 448.936,A -85,B 0,C 180,E1 -26540,E2 -26540} C_VEL
LIN {X 0,Y 103.173,Z 443.374,A -85,B 0,C 180,E1 -26544.136,E2 -26544.136} C_VEL
LIN {X 0,Y 105.482,Z 436.727,A -85,B 0,C 180,E1 -26548.047,E2 -26548.047} C_VEL
LIN {X 0,Y 107.952,Z 429.48,A -85,B 0,C 180,E1 -26551.399,E2 -26551.399} C_VEL
LIN {X 0,Y 110.685,Z 420.749,A -85,B 0,C 180,E1 -26554.552,E2 -26554.552} C_VEL
LIN {X 0,Y 113.675,Z 409.639,A -85,B 0,C 180,E1 -26557.464,E2 -26557.464} C_VEL
LIN {X 0,Y 115.508,Z 400.761,A -85,B 0,C 180,E1 -26559.19,E2 -26559.19} C_VEL
LIN {X 0,Y 116.988,Z 391.694,A -85,B 0,C 180,E1 -26560.487,E2 -26560.487} C_VEL
LIN {X 0,Y 118.127,Z 382.489,A -85,B 0,C 180,E1 -26561.375,E2 -26561.375} C_VEL
LIN {X 0,Y 120.105,Z 354.004,A -85,B 0,C 180,E1 -26563.085,E2 -26563.085} C_VEL
LIN {X 0,Y 112.763,Z 338.241,A -85,B 0,C 180,E1 -26566.779,E2 -26566.779} C_VEL
LIN {X 0,Y 105.402,Z 325.78,A -85,B 0,C 180,E1 -26570.835,E2 -26570.835} C_VEL
LIN {X 0,Y 102.846,Z 321.779,A -85,B 0,C 180,E1 -26572.39,E2 -26572.39} C_VEL
LIN {X 0,Y 101.154,Z 319.081,A -85,B 0,C 180,E1 -26573.49,E2 -26573.49} C_VEL
LIN {X 0,Y 100.834,Z 317.708,A -85,B 0,C 180,E1 -26573.839,E2 -26573.839} C_VEL
LIN {X 0,Y 100.662,Z 317.763,A -85,B 0,C 180,E1 -26579.256,E2 -26579.256} C_VEL
LIN {X 0,Y 100.666,Z 317.748,A -85,B 0,C 180,E1 -26583.952,E2 -26583.952} C_VEL
LIN {X 0,Y 100.648,Z 317.751,A -85,B 0,C 180,E1 -26589.815,E2 -26589.815} C_VEL
LIN {X 0,Y 100.68,Z 317.749,A -85,B 0,C 180,E1 -26595.728,E2 -26595.728} C_VEL
LIN {X 0,Y 100.683,Z 317.746,A -85,B 0,C 180,E1 -26601.08,E2 -26601.08} C_VEL
LIN {X 0,Y 100.701,Z 317.729,A -85,B 0,C 180,E1 -26606.874,E2 -26606.874} C_VEL
LIN {X 0,Y 100.785,Z 317.73,A -85,B 0,C 180,E1 -26615.266,E2 -26615.266} C_VEL
LIN {X 0,Y 100.813,Z 317.701,A -85,B 0,C 180,E1 -26619.6,E2 -26619.6} C_VEL
LIN {X 0,Y 101.101,Z 317.704,A -85,B 0,C 180,E1 -26626.699,E2 -26626.699} C_VEL
LIN {X 0,Y 101.238,Z 317.664,A -85,B 0,C 180,E1 -26632.019,E2 -26632.019} C_VEL
LIN {X 0,Y 101.861,Z 317.602,A -85,B 0,C 180,E1 -26640,E2 -26640} C_VEL
LIN {X 0,Y 101.238,Z 317.66,A -85,B 0,C 180,E1 -26647.98,E2 -26647.98} C_VEL
LIN {X 0,Y 101.101,Z 317.696,A -85,B 0,C 180,E1 -26653.3,E2 -26653.3} C_VEL
LIN {X 0,Y 100.811,Z 317.72,A -85,B 0,C 180,E1 -26660.4,E2 -26660.4} C_VEL
LIN {X 0,Y 100.772,Z 317.743,A -85,B 0,C 180,E1 -26664.959,E2 -26664.959} C_VEL
LIN {X 0,Y 100.686,Z 317.754,A -85,B 0,C 180,E1 -26673.113,E2 -26673.113} C_VEL
LIN {X 0,Y 100.649,Z 317.743,A -85,B 0,C 180,E1 -26677.66,E2 -26677.66} C_VEL
LIN {X 0,Y 101.627,Z 320.573,A -85,B 0,C 180,E1 -26678.491,E2 -26678.491} C_VEL
LIN {X 0,Y 103.5,Z 323.096,A -85,B 0,C 180,E1 -26679.64,E2 -26679.64} C_VEL
LIN {X 0,Y 109.49,Z 333.076,A -85,B 0,C 180,E1 -26683.125,E2 -26683.125} C_VEL
LIN {X 0,Y 113.632,Z 341.086,A -85,B 0,C 180,E1 -26685.376,E2 -26685.376} C_VEL
LIN {X 0,Y 118.222,Z 354.473,A -85,B 0,C 180,E1 -26687.976,E2 -26687.976} C_VEL
LIN {X 0,Y 119.31,Z 369.384,A -85,B 0,C 180,E1 -26689.451,E2 -26689.451} C_VEL
LIN {X 0,Y 117.735,Z 390.35,A -85,B 0,C 180,E1 -26690.766,E2 -26690.766} C_VEL
LIN {X 0,Y 115.912,Z 402.384,A -85,B 0,C 180,E1 -26692.098,E2 -26692.098} C_VEL
LIN {X 0,Y 113.781,Z 412.251,A -85,B 0,C 180,E1 -26693.772,E2 -26693.772} C_VEL
LIN {X 0,Y 111.976,Z 420.136,A -85,B 0,C 180,E1 -26695.608,E2 -26695.608} C_VEL
LIN {X 0,Y 109.38,Z 428.381,A -85,B 0,C 180,E1 -26697.99,E2 -26697.99} C_VEL
LIN {X 0,Y 106.976,Z 436.3,A -85,B 0,C 180,E1 -26701.02,E2 -26701.02} C_VEL
LIN {X 0,Y 104.713,Z 442.811,A -85,B 0,C 180,E1 -26704.135,E2 -26704.135} C_VEL
LIN {X 0,Y 102.545,Z 449.012,A -85,B 0,C 180,E1 -26707.856,E2 -26707.856} C_VEL
LIN {X 0,Y 100.845,Z 454.155,A -85,B 0,C 180,E1 -26711.724,E2 -26711.724} C_VEL
LIN {X 0,Y 99.543,Z 458.418,A -85,B 0,C 180,E1 -26715.694,E2 -26715.694} C_VEL
LIN {X 0,Y 98.668,Z 461.939,A -85,B 0,C 180,E1 -26719.743,E2 -26719.743} C_VEL
LIN {X 0,Y 98.094,Z 465.956,A -85,B 0,C 180,E1 -26725.892,E2 -26725.892} C_VEL
LIN {X 0,Y 98.138,Z 467.889,A -85,B 0,C 180,E1 -26730,E2 -26730} C_VEL
LIN {X 0,Y 98.054,Z 469.285,A -85,B 0,C 180,E1 -26734.11,E2 -26734.11} C_VEL
LIN {X 0,Y 98.327,Z 470.172,A -85,B 0,C 180,E1 -26738.218,E2 -26738.218} C_VEL
LIN {X 0,Y 99.039,Z 470.48,A -85,B 0,C 180,E1 -26742.291,E2 -26742.291} C_VEL
LIN {X 0,Y 100.241,Z 470.34,A -85,B 0,C 180,E1 -26746.286,E2 -26746.286} C_VEL
LIN {X 0,Y 101.885,Z 469.766,A -85,B 0,C 180,E1 -26750.175,E2 -26750.175} C_VEL
LIN {X 0,Y 103.972,Z 468.731,A -85,B 0,C 180,E1 -26753.926,E2 -26753.926} C_VEL
LIN {X 0,Y 107.963,Z 466.13,A -85,B 0,C 180,E1 -26759.223,E2 -26759.223} C_VEL
LIN {X 0,Y 112.95,Z 462.303,A -85,B 0,C 180,E1 -26764.054,E2 -26764.054} C_VEL
LIN {X 0,Y 118.674,Z 457.142,A -85,B 0,C 180,E1 -26768.448,E2 -26768.448} C_VEL
LIN {X 0,Y 125.053,Z 450.414,A -85,B 0,C 180,E1 -26772.406,E2 -26772.406} C_VEL
LIN {X 0,Y 130.768,Z 443.122,A -85,B 0,C 180,E1 -26775.405,E2 -26775.405} C_VEL
LIN {X 0,Y 135.15,Z 436.928,A -85,B 0,C 180,E1 -26777.272,E2 -26777.272} C_VEL
LIN {X 0,Y 139.499,Z 429.569,A -85,B 0,C 180,E1 -26779.085,E2 -26779.085} C_VEL
LIN {X 0,Y 143.459,Z 421.896,A -85,B 0,C 180,E1 -26780.494,E2 -26780.494} C_VEL
LIN {X 0,Y 146.864,Z 414.08,A -85,B 0,C 180,E1 -26781.59,E2 -26781.59} C_VEL
LIN {X 0,Y 149.968,Z 405.206,A -85,B 0,C 180,E1 -26782.534,E2 -26782.534} C_VEL
LIN {X 0,Y 152.448,Z 395.658,A -85,B 0,C 180,E1 -26783.31,E2 -26783.31} C_VEL
LIN {X 0,Y 154.252,Z 385.896,A -85,B 0,C 180,E1 -26783.795,E2 -26783.795} C_VEL
LIN {X 0,Y 154.004,Z 384.407,A -85,B 0,C 180,E1 -26784.224,E2 -26784.224} C_VEL
LIN {X 0,Y 151.793,Z 377.729,A -85,B 0,C 180,E1 -26787.03,E2 -26787.03} C_VEL
LIN {X 0,Y 149.794,Z 372.786,A -85,B 0,C 180,E1 -26789.833,E2 -26789.833} C_VEL
LIN {X 0,Y 147.713,Z 369.095,A -85,B 0,C 180,E1 -26793.128,E2 -26793.128} C_VEL
LIN {X 0,Y 145.829,Z 365.584,A -85,B 0,C 180,E1 -26797.323,E2 -26797.323} C_VEL
LIN {X 0,Y 144.21,Z 362.991,A -85,B 0,C 180,E1 -26804.959,E2 -26804.959} C_VEL
LIN {X 0,Y 144.161,Z 363.036,A -85,B 0,C 180,E1 -26806.511,E2 -26806.511} C_VEL
LIN {X 0,Y 144.152,Z 364.364,A -85,B 0,C 180,E1 -26808.794,E2 -26808.794} C_VEL
LIN {X 0,Y 144.233,Z 366.657,A -85,B 0,C 180,E1 -26810.974,E2 -26810.974} C_VEL
LIN {X 0,Y 144.619,Z 370.42,A -85,B 0,C 180,E1 -26813.855,E2 -26813.855} C_VEL
LIN {X 0,Y 145.496,Z 373.78,A -85,B 0,C 180,E1 -26816.773,E2 -26816.773} C_VEL
LIN {X 0,Y 147.157,Z 376.885,A -85,B 0,C 180,E1 -26820.109,E2 -26820.109} C_VEL
LIN {X 0,Y 149.4,Z 381.861,A -85,B 0,C 180,E1 -26823.756,E2 -26823.756} C_VEL
LIN {X 0,Y 151.005,Z 385.891,A -85,B 0,C 180,E1 -26826.108,E2 -26826.108} C_VEL
LIN {X 0,Y 148.663,Z 397.147,A -85,B 0,C 180,E1 -26826.909,E2 -26826.909} C_VEL
LIN {X 0,Y 145.132,Z 408.109,A -85,B 0,C 180,E1 -26828.036,E2 -26828.036} C_VEL
LIN {X 0,Y 141.528,Z 416.826,A -85,B 0,C 180,E1 -26829.277,E2 -26829.277} C_VEL
LIN {X 0,Y 137.653,Z 424.43,A -85,B 0,C 180,E1 -26830.644,E2 -26830.644} C_VEL
LIN {X 0,Y 133.073,Z 431.976,A -85,B 0,C 180,E1 -26832.389,E2 -26832.389} C_VEL
LIN {X 0,Y 128.712,Z 438.176,A -85,B 0,C 180,E1 -26834.266,E2 -26834.266} C_VEL
LIN {X 0,Y 122.91,Z 445.254,A -85,B 0,C 180,E1 -26837.061,E2 -26837.061} C_VEL
LIN {X 0,Y 116.878,Z 451.472,A -85,B 0,C 180,E1 -26840.408,E2 -26840.408} C_VEL
LIN {X 0,Y 111.526,Z 456.143,A -85,B 0,C 180,E1 -26843.977,E2 -26843.977} C_VEL
LIN {X 0,Y 107.426,Z 459.267,A -85,B 0,C 180,E1 -26847.256,E2 -26847.256} C_VEL
LIN {X 0,Y 103.008,Z 462.129,A -85,B 0,C 180,E1 -26851.48,E2 -26851.48} C_VEL
LIN {X 0,Y 97.91,Z 464.604,A -85,B 0,C 180,E1 -26857.856,E2 -26857.856} C_VEL
LIN {X 0,Y 95.24,Z 465.472,A -85,B 0,C 180,E1 -26862.447,E2 -26862.447} C_VEL
LIN {X 0,Y 93.142,Z 465.699,A -85,B 0,C 180,E1 -26867.229,E2 -26867.229} C_VEL
LIN {X 0,Y 91.679,Z 465.26,A -85,B 0,C 180,E1 -26872.175,E2 -26872.175} C_VEL
LIN {X 0,Y 90.651,Z 463.765,A -85,B 0,C 180,E1 -26878.519,E2 -26878.519} C_VEL
LIN {X 0,Y 90.628,Z 461.269,A -85,B 0,C 180,E1 -26884.754,E2 -26884.754} C_VEL
LIN {X 0,Y 91.301,Z 458.265,A -85,B 0,C 180,E1 -26890.09,E2 -26890.09} C_VEL
LIN {X 0,Y 92.545,Z 453.998,A -85,B 0,C 180,E1 -26895.712,E2 -26895.712} C_VEL
LIN {X 0,Y 94.484,Z 448.228,A -85,B 0,C 180,E1 -26901.445,E2 -26901.445} C_VEL
LIN {X 0,Y 96.652,Z 442.487,A -85,B 0,C 180,E1 -26905.83,E2 -26905.83} C_VEL
LIN {X 0,Y 99.231,Z 435.533,A -85,B 0,C 180,E1 -26910,E2 -26910} C_VEL
LIN {X 0,Y 102.687,Z 425.675,A -85,B 0,C 180,E1 -26914.416,E2 -26914.416} C_VEL
LIN {X 0,Y 105.299,Z 417.306,A -85,B 0,C 180,E1 -26917.189,E2 -26917.189} C_VEL
LIN {X 0,Y 107.831,Z 407.831,A -85,B 0,C 180,E1 -26919.569,E2 -26919.569} C_VEL
LIN {X 0,Y 109.759,Z 398.278,A -85,B 0,C 180,E1 -26921.386,E2 -26921.386} C_VEL
LIN {X 0,Y 111.59,Z 386.598,A -85,B 0,C 180,E1 -26922.897,E2 -26922.897} C_VEL
LIN {X 0,Y 113.061,Z 370.582,A -85,B 0,C 180,E1 -26923.973,E2 -26923.973} C_VEL
LIN {X 0,Y 114.032,Z 356.069,A -85,B 0,C 180,E1 -26924.842,E2 -26924.842} C_VEL
LIN {X 0,Y 107.611,Z 342.032,A -85,B 0,C 180,E1 -26928.415,E2 -26928.415} C_VEL
LIN {X 0,Y 100.721,Z 330.193,A -85,B 0,C 180,E1 -26932.572,E2 -26932.572} C_VEL
LIN {X 0,Y 98.474,Z 326.625,A -85,B 0,C 180,E1 -26934.084,E2 -26934.084} C_VEL
LIN {X 0,Y 96.306,Z 323.285,A -85,B 0,C 180,E1 -26935.636,E2 -26935.636} C_VEL
LIN {X 0,Y 94.378,Z 321.061,A -85,B 0,C 180,E1 -26937.007,E2 -26937.007} C_VEL
LIN {X 0,Y 93.602,Z 318.645,A -85,B 0,C 180,E1 -26937.821,E2 -26937.821} C_VEL
LIN {X 0,Y 93.589,Z 318.631,A -85,B 0,C 180,E1 -26944.305,E2 -26944.305} C_VEL
LIN {X 0,Y 93.548,Z 318.621,A -85,B 0,C 180,E1 -26952.542,E2 -26952.542} C_VEL
LIN {X 0,Y 93.575,Z 318.641,A -85,B 0,C 180,E1 -26958.68,E2 -26958.68} C_VEL
LIN {X 0,Y 93.606,Z 318.605,A -85,B 0,C 180,E1 -26965.676,E2 -26965.676} C_VEL
LIN {X 0,Y 93.667,Z 318.622,A -85,B 0,C 180,E1 -26974.204,E2 -26974.204} C_VEL
LIN {X 0,Y 93.689,Z 318.59,A -85,B 0,C 180,E1 -26977.971,E2 -26977.971} C_VEL
LIN {X 0,Y 94.021,Z 318.585,A -85,B 0,C 180,E1 -26986.339,E2 -26986.339} C_VEL
LIN {X 0,Y 94.172,Z 318.548,A -85,B 0,C 180,E1 -26991.415,E2 -26991.415} C_VEL
LIN {X 0,Y 94.786,Z 318.482,A -85,B 0,C 180,E1 -26999.999,E2 -26999.999} C_VEL
LIN {X 0,Y 94.172,Z 318.536,A -85,B 0,C 180,E1 -27008.583,E2 -27008.583} C_VEL
LIN {X 0,Y 94.021,Z 318.579,A -85,B 0,C 180,E1 -27013.66,E2 -27013.66} C_VEL
LIN {X 0,Y 93.688,Z 318.606,A -85,B 0,C 180,E1 -27022.028,E2 -27022.028} C_VEL
LIN {X 0,Y 93.617,Z 318.636,A -85,B 0,C 180,E1 -27026.771,E2 -27026.771} C_VEL
LIN {X 0,Y 93.625,Z 318.637,A -85,B 0,C 180,E1 -27033.808,E2 -27033.808} C_VEL
LIN {X 0,Y 94.635,Z 321.556,A -85,B 0,C 180,E1 -27034.8,E2 -27034.8} C_VEL
LIN {X 0,Y 96.627,Z 323.977,A -85,B 0,C 180,E1 -27036.224,E2 -27036.224} C_VEL
LIN {X 0,Y 103.157,Z 334.595,A -85,B 0,C 180,E1 -27040.606,E2 -27040.606} C_VEL
LIN {X 0,Y 108.39,Z 344.739,A -85,B 0,C 180,E1 -27043.734,E2 -27043.734} C_VEL
LIN {X 0,Y 112.335,Z 356.599,A -85,B 0,C 180,E1 -27046.222,E2 -27046.222} C_VEL
LIN {X 0,Y 113.265,Z 369.685,A -85,B 0,C 180,E1 -27047.621,E2 -27047.621} C_VEL
LIN {X 0,Y 111.625,Z 390.32,A -85,B 0,C 180,E1 -27048.966,E2 -27048.966} C_VEL
LIN {X 0,Y 109.862,Z 401.574,A -85,B 0,C 180,E1 -27050.231,E2 -27050.231} C_VEL
LIN {X 0,Y 107.442,Z 412.293,A -85,B 0,C 180,E1 -27052.116,E2 -27052.116} C_VEL
LIN {X 0,Y 105.749,Z 419.476,A -85,B 0,C 180,E1 -27053.857,E2 -27053.857} C_VEL
LIN {X 0,Y 103.012,Z 427.802,A -85,B 0,C 180,E1 -27056.337,E2 -27056.337} C_VEL
LIN {X 0,Y 100.456,Z 435.787,A -85,B 0,C 180,E1 -27059.522,E2 -27059.522} C_VEL
LIN {X 0,Y 97.721,Z 443.203,A -85,B 0,C 180,E1 -27063.29,E2 -27063.29} C_VEL
LIN {X 0,Y 95.007,Z 450.737,A -85,B 0,C 180,E1 -27068.293,E2 -27068.293} C_VEL
LIN {X 0,Y 92.664,Z 457.588,A -85,B 0,C 180,E1 -27074.606,E2 -27074.606} C_VEL
LIN {X 0,Y 91.346,Z 462.761,A -85,B 0,C 180,E1 -27081.149,E2 -27081.149} C_VEL
LIN {X 0,Y 90.966,Z 466.522,A -85,B 0,C 180,E1 -27087.786,E2 -27087.786} C_VEL
LIN {X 0,Y 91.045,Z 467.426,A -85,B 0,C 180,E1 -27090,E2 -27090} C_VEL
LIN {X 0,Y 90.982,Z 468.923,A -85,B 0,C 180,E1 -27094.43,E2 -27094.43} C_VEL
LIN {X 0,Y 91.31,Z 469.826,A -85,B 0,C 180,E1 -27098.855,E2 -27098.855} C_VEL
LIN {X 0,Y 92.108,Z 470.227,A -85,B 0,C 180,E1 -27103.232,E2 -27103.232} C_VEL
LIN {X 0,Y 93.438,Z 470.198,A -85,B 0,C 180,E1 -27107.509,E2 -27107.509} C_VEL
LIN {X 0,Y 95.251,Z 469.738,A -85,B 0,C 180,E1 -27111.648,E2 -27111.648} C_VEL
LIN {X 0,Y 97.504,Z 468.736,A -85,B 0,C 180,E1 -27115.624,E2 -27115.624} C_VEL
LIN {X 0,Y 101.831,Z 466.329,A -85,B 0,C 180,E1 -27121.172,E2 -27121.172} C_VEL
LIN {X 0,Y 107.157,Z 462.644,A -85,B 0,C 180,E1 -27126.175,E2 -27126.175} C_VEL
LIN {X 0,Y 111.146,Z 459.523,A -85,B 0,C 180,E1 -27129.22,E2 -27129.22} C_VEL
LIN {X 0,Y 116.567,Z 454.593,A -85,B 0,C 180,E1 -27132.708,E2 -27132.708} C_VEL
LIN {X 0,Y 121.17,Z 449.847,A -85,B 0,C 180,E1 -27135.275,E2 -27135.275} C_VEL
LIN {X 0,Y 127.198,Z 442.503,A -85,B 0,C 180,E1 -27138.235,E2 -27138.235} C_VEL
LIN {X 0,Y 131.746,Z 436.275,A -85,B 0,C 180,E1 -27140.067,E2 -27140.067} C_VEL
LIN {X 0,Y 136.237,Z 429.048,A -85,B 0,C 180,E1 -27141.755,E2 -27141.755} C_VEL
LIN {X 0,Y 140.509,Z 421.006,A -85,B 0,C 180,E1 -27143.156,E2 -27143.156} C_VEL
LIN {X 0,Y 144.033,Z 413.03,A -85,B 0,C 180,E1 -27144.211,E2 -27144.211} C_VEL
LIN {X 0,Y 147.299,Z 403.775,A -85,B 0,C 180,E1 -27145.124,E2 -27145.124} C_VEL
LIN {X 0,Y 149.754,Z 394.308,A -85,B 0,C 180,E1 -27145.835,E2 -27145.835} C_VEL
LIN {X 0,Y 150.891,Z 388.385,A -85,B 0,C 180,E1 -27146.163,E2 -27146.163} C_VEL
LIN {X 0,Y 148.905,Z 381.506,A -85,B 0,C 180,E1 -27149.413,E2 -27149.413} C_VEL
LIN {X 0,Y 147.775,Z 378.754,A -85,B 0,C 180,E1 -27151.215,E2 -27151.215} C_VEL
LIN {X 0,Y 146.117,Z 375.558,A -85,B 0,C 180,E1 -27154.158,E2 -27154.158} C_VEL
LIN {X 0,Y 144.755,Z 372.554,A -85,B 0,C 180,E1 -27157.552,E2 -27157.552} C_VEL
LIN {X 0,Y 143.221,Z 369.857,A -85,B 0,C 180,E1 -27165.798,E2 -27165.798} C_VEL
LIN {X 0,Y 143.415,Z 370.075,A -85,B 0,C 180,E1 -27169.134,E2 -27169.134} C_VEL
LIN {X 0,Y 145.016,Z 372.422,A -85,B 0,C 180,E1 -27175.446,E2 -27175.446} C_VEL
LIN {X 0,Y 145.496,Z 373.78,A -85,B 0,C 180,E1 -27176.773,E2 -27176.773} C_VEL
LIN {X 0,Y 145.987,Z 375.733,A -85,B 0,C 180,E1 -27178.103,E2 -27178.103} C_VEL
LIN {X 0,Y 146.455,Z 380.552,A -85,B 0,C 180,E1 -27179.899,E2 -27179.899} C_VEL
LIN {X 0,Y 146.95,Z 386.68,A -85,B 0,C 180,E1 -27182.003,E2 -27182.003} C_VEL
LIN {X 0,Y 147.293,Z 388.29,A -85,B 0,C 180,E1 -27182.839,E2 -27182.839} C_VEL
LIN {X 0,Y 147.732,Z 389.793,A -85,B 0,C 180,E1 -27183.798,E2 -27183.798} C_VEL
LIN {X 0,Y 145.08,Z 400.203,A -85,B 0,C 180,E1 -27184.607,E2 -27184.607} C_VEL
LIN {X 0,Y 141.93,Z 409.237,A -85,B 0,C 180,E1 -27185.552,E2 -27185.552} C_VEL
LIN {X 0,Y 138.01,Z 418.086,A -85,B 0,C 180,E1 -27186.792,E2 -27186.792} C_VEL
LIN {X 0,Y 132.963,Z 427.243,A -85,B 0,C 180,E1 -27188.46,E2 -27188.46} C_VEL
LIN {X 0,Y 126.96,Z 436.083,A -85,B 0,C 180,E1 -27190.724,E2 -27190.724} C_VEL
LIN {X 0,Y 120.523,Z 443.813,A -85,B 0,C 180,E1 -27193.489,E2 -27193.489} C_VEL
LIN {X 0,Y 113.822,Z 450.566,A -85,B 0,C 180,E1 -27196.859,E2 -27196.859} C_VEL
LIN {X 0,Y 108.422,Z 455.159,A -85,B 0,C 180,E1 -27200.08,E2 -27200.08} C_VEL
LIN {X 0,Y 101.178,Z 460.262,A -85,B 0,C 180,E1 -27205.448,E2 -27205.448} C_VEL
LIN {X 0,Y 95.433,Z 463.374,A -85,B 0,C 180,E1 -27211.032,E2 -27211.032} C_VEL
LIN {X 0,Y 93.089,Z 464.468,A -85,B 0,C 180,E1 -27213.856,E2 -27213.856} C_VEL
LIN {X 0,Y 89.763,Z 465.555,A -85,B 0,C 180,E1 -27218.783,E2 -27218.783} C_VEL
LIN {X 0,Y 87.297,Z 465.891,A -85,B 0,C 180,E1 -27223.569,E2 -27223.569} C_VEL
LIN {X 0,Y 85.362,Z 465.619,A -85,B 0,C 180,E1 -27228.805,E2 -27228.805} C_VEL
LIN {X 0,Y 83.672,Z 464.041,A -85,B 0,C 180,E1 -27237.136,E2 -27237.136} C_VEL
LIN {X 0,Y 83.42,Z 462.24,A -85,B 0,C 180,E1 -27242.396,E2 -27242.396} C_VEL
LIN {X 0,Y 84.231,Z 458.094,A -85,B 0,C 180,E1 -27250.504,E2 -27250.504} C_VEL
LIN {X 0,Y 85.773,Z 453.185,A -85,B 0,C 180,E1 -27257.245,E2 -27257.245} C_VEL
LIN {X 0,Y 87.354,Z 448.769,A -85,B 0,C 180,E1 -27261.906,E2 -27261.906} C_VEL
LIN {X 0,Y 89.633,Z 443.097,A -85,B 0,C 180,E1 -27266.63,E2 -27266.63} C_VEL
LIN {X 0,Y 92.317,Z 436.24,A -85,B 0,C 180,E1 -27271.091,E2 -27271.091} C_VEL
LIN {X 0,Y 95.513,Z 427.827,A -85,B 0,C 180,E1 -27275.277,E2 -27275.277} C_VEL
LIN {X 0,Y 98.729,Z 418.341,A -85,B 0,C 180,E1 -27278.719,E2 -27278.719} C_VEL
LIN {X 0,Y 101.455,Z 408.734,A -85,B 0,C 180,E1 -27281.297,E2 -27281.297} C_VEL
LIN {X 0,Y 103.395,Z 400.152,A -85,B 0,C 180,E1 -27283.039,E2 -27283.039} C_VEL
LIN {X 0,Y 105.062,Z 390.619,A -85,B 0,C 180,E1 -27284.446,E2 -27284.446} C_VEL
LIN {X 0,Y 106.367,Z 379.946,A -85,B 0,C 180,E1 -27285.461,E2 -27285.461} C_VEL
LIN {X 0,Y 107.998,Z 358.049,A -85,B 0,C 180,E1 -27286.836,E2 -27286.836} C_VEL
LIN {X 0,Y 102.799,Z 346.359,A -85,B 0,C 180,E1 -27290.009,E2 -27290.009} C_VEL
LIN {X 0,Y 96.376,Z 334.964,A -85,B 0,C 180,E1 -27294.311,E2 -27294.311} C_VEL
LIN {X 0,Y 92.394,Z 328.717,A -85,B 0,C 180,E1 -27297.302,E2 -27297.302} C_VEL
LIN {X 0,Y 90.055,Z 325.456,A -85,B 0,C 180,E1 -27299.198,E2 -27299.198} C_VEL
LIN {X 0,Y 89.21,Z 324.193,A -85,B 0,C 180,E1 -27299.935,E2 -27299.935} C_VEL
LIN {X 0,Y 87.313,Z 321.96,A -85,B 0,C 180,E1 -27301.599,E2 -27301.599} C_VEL
LIN {X 0,Y 86.542,Z 319.504,A -85,B 0,C 180,E1 -27302.682,E2 -27302.682} C_VEL
LIN {X 0,Y 86.465,Z 319.509,A -85,B 0,C 180,E1 -27310.559,E2 -27310.559} C_VEL
LIN {X 0,Y 86.504,Z 319.52,A -85,B 0,C 180,E1 -27316.985,E2 -27316.985} C_VEL
LIN {X 0,Y 86.554,Z 319.482,A -85,B 0,C 180,E1 -27325.361,E2 -27325.361} C_VEL
LIN {X 0,Y 86.583,Z 319.509,A -85,B 0,C 180,E1 -27333.234,E2 -27333.234} C_VEL
LIN {X 0,Y 86.642,Z 319.468,A -85,B 0,C 180,E1 -27341.066,E2 -27341.066} C_VEL
LIN {X 0,Y 86.929,Z 319.468,A -85,B 0,C 180,E1 -27345.963,E2 -27345.963} C_VEL
LIN {X 0,Y 87.082,Z 319.436,A -85,B 0,C 180,E1 -27350.711,E2 -27350.711} C_VEL
LIN {X 0,Y 87.712,Z 319.362,A -85,B 0,C 180,E1 -27359.999,E2 -27359.999} C_VEL
LIN {X 0,Y 87.081,Z 319.417,A -85,B 0,C 180,E1 -27369.288,E2 -27369.288} C_VEL
LIN {X 0,Y 86.929,Z 319.464,A -85,B 0,C 180,E1 -27374.036,E2 -27374.036} C_VEL
LIN {X 0,Y 86.641,Z 319.491,A -85,B 0,C 180,E1 -27378.933,E2 -27378.933} C_VEL
LIN {X 0,Y 86.581,Z 319.513,A -85,B 0,C 180,E1 -27386.763,E2 -27386.763} C_VEL
LIN {X 0,Y 86.497,Z 319.656,A -85,B 0,C 180,E1 -27389.077,E2 -27389.077} C_VEL
LIN {X 0,Y 87.44,Z 322.311,A -85,B 0,C 180,E1 -27390.154,E2 -27390.154} C_VEL
LIN {X 0,Y 89.839,Z 325.001,A -85,B 0,C 180,E1 -27392.203,E2 -27392.203} C_VEL
LIN {X 0,Y 91.982,Z 328.361,A -85,B 0,C 180,E1 -27394,E2 -27394} C_VEL
LIN {X 0,Y 96.916,Z 336.235,A -85,B 0,C 180,E1 -27397.723,E2 -27397.723} C_VEL
LIN {X 0,Y 102.626,Z 346.929,A -85,B 0,C 180,E1 -27401.565,E2 -27401.565} C_VEL
LIN {X 0,Y 105.857,Z 356.227,A -85,B 0,C 180,E1 -27403.775,E2 -27403.775} C_VEL
LIN {X 0,Y 106.778,Z 359.615,A -85,B 0,C 180,E1 -27404.443,E2 -27404.443} C_VEL
LIN {X 0,Y 107.297,Z 370.704,A -85,B 0,C 180,E1 -27405.632,E2 -27405.632} C_VEL
LIN {X 0,Y 105.607,Z 390.63,A -85,B 0,C 180,E1 -27406.99,E2 -27406.99} C_VEL
LIN {X 0,Y 103.518,Z 402.661,A -85,B 0,C 180,E1 -27408.46,E2 -27408.46} C_VEL
LIN {X 0,Y 101.365,Z 411.686,A -85,B 0,C 180,E1 -27410.104,E2 -27410.104} C_VEL
LIN {X 0,Y 99.615,Z 418.809,A -85,B 0,C 180,E1 -27411.88,E2 -27411.88} C_VEL
LIN {X 0,Y 96.742,Z 427.223,A -85,B 0,C 180,E1 -27414.468,E2 -27414.468} C_VEL
LIN {X 0,Y 94.015,Z 435.273,A -85,B 0,C 180,E1 -27417.818,E2 -27417.818} C_VEL
LIN {X 0,Y 91.414,Z 441.88,A -85,B 0,C 180,E1 -27421.282,E2 -27421.282} C_VEL
LIN {X 0,Y 88.948,Z 448.166,A -85,B 0,C 180,E1 -27425.493,E2 -27425.493} C_VEL
LIN {X 0,Y 86.996,Z 453.382,A -85,B 0,C 180,E1 -27429.92,E2 -27429.92} C_VEL
LIN {X 0,Y 85.219,Z 458.67,A -85,B 0,C 180,E1 -27435.676,E2 -27435.676} C_VEL
LIN {X 0,Y 84.348,Z 462.049,A -85,B 0,C 180,E1 -27440.408,E2 -27440.408} C_VEL
LIN {X 0,Y 83.97,Z 464.789,A -85,B 0,C 180,E1 -27445.199,E2 -27445.199} C_VEL
LIN {X 0,Y 83.963,Z 466.949,A -85,B 0,C 180,E1 -27450,E2 -27450} C_VEL
LIN {X 0,Y 83.931,Z 468.494,A -85,B 0,C 180,E1 -27454.803,E2 -27454.803} C_VEL
LIN {X 0,Y 84.318,Z 469.457,A -85,B 0,C 180,E1 -27459.596,E2 -27459.596} C_VEL
LIN {X 0,Y 85.216,Z 469.972,A -85,B 0,C 180,E1 -27464.324,E2 -27464.324} C_VEL
LIN {X 0,Y 86.692,Z 470.058,A -85,B 0,C 180,E1 -27468.921,E2 -27468.921} C_VEL
LIN {X 0,Y 88.674,Z 469.671,A -85,B 0,C 180,E1 -27473.345,E2 -27473.345} C_VEL
LIN {X 0,Y 91.134,Z 468.71,A -85,B 0,C 180,E1 -27477.561,E2 -27477.561} C_VEL
LIN {X 0,Y 94.126,Z 467.29,A -85,B 0,C 180,E1 -27481.51,E2 -27481.51} C_VEL
LIN {X 0,Y 99.543,Z 464.247,A -85,B 0,C 180,E1 -27486.877,E2 -27486.877} C_VEL
LIN {X 0,Y 105.769,Z 459.973,A -85,B 0,C 180,E1 -27491.64,E2 -27491.64} C_VEL
LIN {X 0,Y 112.683,Z 454.129,A -85,B 0,C 180,E1 -27495.826,E2 -27495.826} C_VEL
LIN {X 0,Y 118.81,Z 447.935,A -85,B 0,C 180,E1 -27498.954,E2 -27498.954} C_VEL
LIN {X 0,Y 123.968,Z 441.913,A -85,B 0,C 180,E1 -27501.214,E2 -27501.214} C_VEL
LIN {X 0,Y 129.459,Z 434.506,A -85,B 0,C 180,E1 -27503.267,E2 -27503.267} C_VEL
LIN {X 0,Y 134.265,Z 426.84,A -85,B 0,C 180,E1 -27504.868,E2 -27504.868} C_VEL
LIN {X 0,Y 139.339,Z 417.179,A -85,B 0,C 180,E1 -27506.326,E2 -27506.326} C_VEL
LIN {X 0,Y 143.793,Z 406.031,A -85,B 0,C 180,E1 -27507.504,E2 -27507.504} C_VEL
LIN {X 0,Y 146.74,Z 395.751,A -85,B 0,C 180,E1 -27508.286,E2 -27508.286} C_VEL
LIN {X 0,Y 147.707,Z 391.624,A -85,B 0,C 180,E1 -27508.54,E2 -27508.54} C_VEL
LIN {X 0,Y 146.334,Z 386.055,A -85,B 0,C 180,E1 -27511.484,E2 -27511.484} C_VEL
LIN {X 0,Y 144.669,Z 382.131,A -85,B 0,C 180,E1 -27515.037,E2 -27515.037} C_VEL
LIN {X 0,Y 143.357,Z 379.28,A -85,B 0,C 180,E1 -27518.659,E2 -27518.659} C_VEL
LIN {X 0,Y 142.254,Z 376.931,A -85,B 0,C 180,E1 -27525.699,E2 -27525.699} C_VEL
LIN {X 0,Y 142.434,Z 377.132,A -85,B 0,C 180,E1 -27529.058,E2 -27529.058} C_VEL
LIN {X 0,Y 143.791,Z 379.412,A -85,B 0,C 180,E1 -27534.899,E2 -27534.899} C_VEL
LIN {X 0,Y 145.476,Z 383.506,A -85,B 0,C 180,E1 -27539.308,E2 -27539.308} C_VEL
LIN {X 0,Y 147.293,Z 388.29,A -85,B 0,C 180,E1 -27542.839,E2 -27542.839} C_VEL
LIN {X 0,Y 147.293,Z 390.071,A -85,B 0,C 180,E1 -27543.373,E2 -27543.373} C_VEL
LIN {X 0,Y 146.634,Z 392.984,A -85,B 0,C 180,E1 -27543.559,E2 -27543.559} C_VEL
LIN {X 0,Y 145.046,Z 397.268,A -85,B 0,C 180,E1 -27543.294,E2 -27543.294} C_VEL
LIN {X 0,Y 141.804,Z 404.166,A -85,B 0,C 180,E1 -27542.629,E2 -27542.629} C_VEL
LIN {X 0,Y 139.922,Z 408.271,A -85,B 0,C 180,E1 -27542.703,E2 -27542.703} C_VEL
LIN {X 0,Y 136.197,Z 416.663,A -85,B 0,C 180,E1 -27543.774,E2 -27543.774} C_VEL
LIN {X 0,Y 132.26,Z 423.924,A -85,B 0,C 180,E1 -27544.939,E2 -27544.939} C_VEL
LIN {X 0,Y 127.323,Z 431.533,A -85,B 0,C 180,E1 -27546.517,E2 -27546.517} C_VEL
LIN {X 0,Y 122.502,Z 437.89,A -85,B 0,C 180,E1 -27548.268,E2 -27548.268} C_VEL
LIN {X 0,Y 117.287,Z 443.79,A -85,B 0,C 180,E1 -27550.356,E2 -27550.356} C_VEL
LIN {X 0,Y 111.729,Z 449.185,A -85,B 0,C 180,E1 -27552.851,E2 -27552.851} C_VEL
LIN {X 0,Y 107.112,Z 453.125,A -85,B 0,C 180,E1 -27555.216,E2 -27555.216} C_VEL
LIN {X 0,Y 103.187,Z 456.161,A -85,B 0,C 180,E1 -27557.542,E2 -27557.542} C_VEL
LIN {X 0,Y 97.918,Z 459.612,A -85,B 0,C 180,E1 -27561.087,E2 -27561.087} C_VEL
LIN {X 0,Y 93.109,Z 462.262,A -85,B 0,C 180,E1 -27565.076,E2 -27565.076} C_VEL
LIN {X 0,Y 88.765,Z 464.176,A -85,B 0,C 180,E1 -27569.437,E2 -27569.437} C_VEL
LIN {X 0,Y 83.868,Z 465.751,A -85,B 0,C 180,E1 -27575.916,E2 -27575.916} C_VEL
LIN {X 0,Y 79.302,Z 465.939,A -85,B 0,C 180,E1 -27585.154,E2 -27585.154} C_VEL
LIN {X 0,Y 77.638,Z 465.284,A -85,B 0,C 180,E1 -27590.681,E2 -27590.681} C_VEL
LIN {X 0,Y 76.616,Z 463.979,A -85,B 0,C 180,E1 -27596.608,E2 -27596.608} C_VEL
LIN {X 0,Y 76.334,Z 462.019,A -85,B 0,C 180,E1 -27602.592,E2 -27602.592} C_VEL
LIN {X 0,Y 76.792,Z 459.35,A -85,B 0,C 180,E1 -27608.527,E2 -27608.527} C_VEL
LIN {X 0,Y 77.784,Z 455.95,A -85,B 0,C 180,E1 -27614.273,E2 -27614.273} C_VEL
LIN {X 0,Y 79.773,Z 450.557,A -85,B 0,C 180,E1 -27621.131,E2 -27621.131} C_VEL
LIN {X 0,Y 81.948,Z 445.225,A -85,B 0,C 180,E1 -27626.312,E2 -27626.312} C_VEL
LIN {X 0,Y 84.9,Z 438.173,A -85,B 0,C 180,E1 -27631.543,E2 -27631.543} C_VEL
LIN {X 0,Y 87.904,Z 430.766,A -85,B 0,C 180,E1 -27635.736,E2 -27635.736} C_VEL
LIN {X 0,Y 90.667,Z 423.486,A -85,B 0,C 180,E1 -27638.918,E2 -27638.918} C_VEL
LIN {X 0,Y 93.731,Z 414.447,A -85,B 0,C 180,E1 -27641.939,E2 -27641.939} C_VEL
LIN {X 0,Y 96.681,Z 403.582,A -85,B 0,C 180,E1 -27644.603,E2 -27644.603} C_VEL
LIN {X 0,Y 98.836,Z 392.729,A -85,B 0,C 180,E1 -27646.39,E2 -27646.39} C_VEL
LIN {X 0,Y 100.183,Z 383.181,A -85,B 0,C 180,E1 -27647.432,E2 -27647.432} C_VEL
LIN {X 0,Y 102.198,Z 360.317,A -85,B 0,C 180,E1 -27648.924,E2 -27648.924} C_VEL
LIN {X 0,Y 97.779,Z 350.061,A -85,B 0,C 180,E1 -27651.968,E2 -27651.968} C_VEL
LIN {X 0,Y 91.702,Z 339.11,A -85,B 0,C 180,E1 -27656.489,E2 -27656.489} C_VEL
LIN {X 0,Y 88.371,Z 333.83,A -85,B 0,C 180,E1 -27659.272,E2 -27659.272} C_VEL
LIN {X 0,Y 85.436,Z 329.601,A -85,B 0,C 180,E1 -27661.982,E2 -27661.982} C_VEL
LIN {X 0,Y 83.277,Z 326.347,A -85,B 0,C 180,E1 -27664.201,E2 -27664.201} C_VEL
LIN {X 0,Y 82.896,Z 325.588,A -85,B 0,C 180,E1 -27664.644,E2 -27664.644} C_VEL
LIN {X 0,Y 80.499,Z 323.412,A -85,B 0,C 180,E1 -27667.187,E2 -27667.187} C_VEL
LIN {X 0,Y 79.492,Z 321.063,A -85,B 0,C 180,E1 -27668.587,E2 -27668.587} C_VEL
LIN {X 0,Y 79.385,Z 320.404,A -85,B 0,C 180,E1 -27668.926,E2 -27668.926} C_VEL
LIN {X 0,Y 79.414,Z 320.389,A -85,B 0,C 180,E1 -27675.069,E2 -27675.069} C_VEL
LIN {X 0,Y 79.406,Z 320.378,A -85,B 0,C 180,E1 -27682.801,E2 -27682.801} C_VEL
LIN {X 0,Y 79.389,Z 320.387,A -85,B 0,C 180,E1 -27687.916,E2 -27687.916} C_VEL
LIN {X 0,Y 79.523,Z 320.385,A -85,B 0,C 180,E1 -27693.775,E2 -27693.775} C_VEL
LIN {X 0,Y 79.51,Z 320.351,A -85,B 0,C 180,E1 -27699.294,E2 -27699.294} C_VEL
LIN {X 0,Y 79.823,Z 320.351,A -85,B 0,C 180,E1 -27705.572,E2 -27705.572} C_VEL
LIN {X 0,Y 79.965,Z 320.327,A -85,B 0,C 180,E1 -27709.875,E2 -27709.875} C_VEL
LIN {X 0,Y 80.639,Z 320.243,A -85,B 0,C 180,E1 -27719.999,E2 -27719.999} C_VEL
LIN {X 0,Y 79.965,Z 320.304,A -85,B 0,C 180,E1 -27730.123,E2 -27730.123} C_VEL
LIN {X 0,Y 79.742,Z 320.364,A -85,B 0,C 180,E1 -27735.331,E2 -27735.331} C_VEL
LIN {X 0,Y 79.515,Z 320.412,A -85,B 0,C 180,E1 -27742.92,E2 -27742.92} C_VEL
LIN {X 0,Y 80.474,Z 323.144,A -85,B 0,C 180,E1 -27744.336,E2 -27744.336} C_VEL
LIN {X 0,Y 82.63,Z 325.413,A -85,B 0,C 180,E1 -27746.699,E2 -27746.699} C_VEL
LIN {X 0,Y 85.273,Z 329.456,A -85,B 0,C 180,E1 -27749.483,E2 -27749.483} C_VEL
LIN {X 0,Y 86.525,Z 331.218,A -85,B 0,C 180,E1 -27750.676,E2 -27750.676} C_VEL
LIN {X 0,Y 90.725,Z 337.651,A -85,B 0,C 180,E1 -27754.335,E2 -27754.335} C_VEL
LIN {X 0,Y 95.611,Z 346.657,A -85,B 0,C 180,E1 -27758.163,E2 -27758.163} C_VEL
LIN {X 0,Y 98.371,Z 352.588,A -85,B 0,C 180,E1 -27760.182,E2 -27760.182} C_VEL
LIN {X 0,Y 100.99,Z 361.025,A -85,B 0,C 180,E1 -27762.221,E2 -27762.221} C_VEL
LIN {X 0,Y 101.524,Z 370.457,A -85,B 0,C 180,E1 -27763.357,E2 -27763.357} C_VEL
LIN {X 0,Y 99.75,Z 390.317,A -85,B 0,C 180,E1 -27764.754,E2 -27764.754} C_VEL
LIN {X 0,Y 97.816,Z 401.366,A -85,B 0,C 180,E1 -27766.095,E2 -27766.095} C_VEL
LIN {X 0,Y 95.244,Z 411.618,A -85,B 0,C 180,E1 -27768.008,E2 -27768.008} C_VEL
LIN {X 0,Y 93.122,Z 419.503,A -85,B 0,C 180,E1 -27770.098,E2 -27770.098} C_VEL
LIN {X 0,Y 90.112,Z 427.745,A -85,B 0,C 180,E1 -27772.813,E2 -27772.813} C_VEL
LIN {X 0,Y 87.233,Z 435.67,A -85,B 0,C 180,E1 -27776.367,E2 -27776.367} C_VEL
LIN {X 0,Y 84.506,Z 442.173,A -85,B 0,C 180,E1 -27780.068,E2 -27780.068} C_VEL
LIN {X 0,Y 81.919,Z 448.377,A -85,B 0,C 180,E1 -27784.599,E2 -27784.599} C_VEL
LIN {X 0,Y 79.895,Z 453.524,A -85,B 0,C 180,E1 -27789.399,E2 -27789.399} C_VEL
LIN {X 0,Y 78.361,Z 457.788,A -85,B 0,C 180,E1 -27794.392,E2 -27794.392} C_VEL
LIN {X 0,Y 77.378,Z 461.31,A -85,B 0,C 180,E1 -27799.534,E2 -27799.534} C_VEL
LIN {X 0,Y 76.83,Z 465.321,A -85,B 0,C 180,E1 -27807.379,E2 -27807.379} C_VEL
LIN {X 0,Y 76.884,Z 466.434,A -85,B 0,C 180,E1 -27810,E2 -27810} C_VEL
LIN {X 0,Y 76.868,Z 468.011,A -85,B 0,C 180,E1 -27815.246,E2 -27815.246} C_VEL
LIN {X 0,Y 77.329,Z 469.087,A -85,B 0,C 180,E1 -27820.472,E2 -27820.472} C_VEL
LIN {X 0,Y 78.341,Z 469.716,A -85,B 0,C 180,E1 -27825.612,E2 -27825.612} C_VEL
LIN {X 0,Y 80.014,Z 469.913,A -85,B 0,C 180,E1 -27830.569,E2 -27830.569} C_VEL
LIN {X 0,Y 82.194,Z 469.546,A -85,B 0,C 180,E1 -27835.31,E2 -27835.31} C_VEL
LIN {X 0,Y 84.886,Z 468.695,A -85,B 0,C 180,E1 -27839.785,E2 -27839.785} C_VEL
LIN {X 0,Y 88.158,Z 467.405,A -85,B 0,C 180,E1 -27843.919,E2 -27843.919} C_VEL
LIN {X 0,Y 93.964,Z 464.493,A -85,B 0,C 180,E1 -27849.474,E2 -27849.474} C_VEL
LIN {X 0,Y 100.588,Z 460.362,A -85,B 0,C 180,E1 -27854.32,E2 -27854.32} C_VEL
LIN {X 0,Y 107.888,Z 454.817,A -85,B 0,C 180,E1 -27858.513,E2 -27858.513} C_VEL
LIN {X 0,Y 114.313,Z 448.824,A -85,B 0,C 180,E1 -27861.614,E2 -27861.614} C_VEL
LIN {X 0,Y 119.683,Z 443.047,A -85,B 0,C 180,E1 -27863.843,E2 -27863.843} C_VEL
LIN {X 0,Y 125.395,Z 435.926,A -85,B 0,C 180,E1 -27865.833,E2 -27865.833} C_VEL
LIN {X 0,Y 130.359,Z 428.617,A -85,B 0,C 180,E1 -27867.387,E2 -27867.387} C_VEL
LIN {X 0,Y 134.83,Z 420.872,A -85,B 0,C 180,E1 -27868.597,E2 -27868.597} C_VEL
LIN {X 0,Y 138.61,Z 412.977,A -85,B 0,C 180,E1 -27869.534,E2 -27869.534} C_VEL
LIN {X 0,Y 142.227,Z 403.404,A -85,B 0,C 180,E1 -27870.387,E2 -27870.387} C_VEL
LIN {X 0,Y 144.559,Z 394.916,A -85,B 0,C 180,E1 -27871.054,E2 -27871.054} C_VEL
LIN {X 0,Y 144.021,Z 391.644,A -85,B 0,C 180,E1 -27873.016,E2 -27873.016} C_VEL
LIN {X 0,Y 142.861,Z 388.369,A -85,B 0,C 180,E1 -27876.248,E2 -27876.248} C_VEL
LIN {X 0,Y 142.083,Z 386.237,A -85,B 0,C 180,E1 -27878.914,E2 -27878.914} C_VEL
LIN {X 0,Y 141.162,Z 383.986,A -85,B 0,C 180,E1 -27885.586,E2 -27885.586} C_VEL
LIN {X 0,Y 141.297,Z 384.202,A -85,B 0,C 180,E1 -27888.955,E2 -27888.955} C_VEL
LIN {X 0,Y 142.3,Z 386.145,A -85,B 0,C 180,E1 -27894.214,E2 -27894.214} C_VEL
LIN {X 0,Y 143.57,Z 390.059,A -85,B 0,C 180,E1 -27898.474,E2 -27898.474} C_VEL
LIN {X 0,Y 144.529,Z 393.977,A -85,B 0,C 180,E1 -27901.458,E2 -27901.458} C_VEL
LIN {X 0,Y 141.115,Z 405.292,A -85,B 0,C 180,E1 -27902.371,E2 -27902.371} C_VEL
LIN {X 0,Y 139.922,Z 408.271,A -85,B 0,C 180,E1 -27902.703,E2 -27902.703} C_VEL
LIN {X 0,Y 137.402,Z 413.749,A -85,B 0,C 180,E1 -27903.041,E2 -27903.041} C_VEL
LIN {X 0,Y 132.056,Z 422.267,A -85,B 0,C 180,E1 -27903.113,E2 -27903.113} C_VEL
LIN {X 0,Y 126.202,Z 430.066,A -85,B 0,C 180,E1 -27903.395,E2 -27903.395} C_VEL
LIN {X 0,Y 122.79,Z 434.37,A -85,B 0,C 180,E1 -27904.099,E2 -27904.099} C_VEL
LIN {X 0,Y 115.344,Z 442.931,A -85,B 0,C 180,E1 -27906.724,E2 -27906.724} C_VEL
LIN {X 0,Y 108.642,Z 449.204,A -85,B 0,C 180,E1 -27909.431,E2 -27909.431} C_VEL
LIN {X 0,Y 103.683,Z 453.22,A -85,B 0,C 180,E1 -27911.733,E2 -27911.733} C_VEL
LIN {X 0,Y 98.112,Z 457.123,A -85,B 0,C 180,E1 -27914.759,E2 -27914.759} C_VEL
LIN {X 0,Y 91.868,Z 460.74,A -85,B 0,C 180,E1 -27918.831,E2 -27918.831} C_VEL
LIN {X 0,Y 85.349,Z 463.72,A -85,B 0,C 180,E1 -27924.314,E2 -27924.314} C_VEL
LIN {X 0,Y 78.249,Z 465.944,A -85,B 0,C 180,E1 -27932.609,E2 -27932.609} C_VEL
LIN {X 0,Y 72.967,Z 466.153,A -85,B 0,C 180,E1 -27942.395,E2 -27942.395} C_VEL
LIN {X 0,Y 71.506,Z 465.826,A -85,B 0,C 180,E1 -27946.53,E2 -27946.53} C_VEL
LIN {X 0,Y 69.907,Z 464.562,A -85,B 0,C 180,E1 -27953.541,E2 -27953.541} C_VEL
LIN {X 0,Y 69.271,Z 461.709,A -85,B 0,C 180,E1 -27962.839,E2 -27962.839} C_VEL
LIN {X 0,Y 69.794,Z 458.913,A -85,B 0,C 180,E1 -27969.364,E2 -27969.364} C_VEL
LIN {X 0,Y 71.344,Z 454.222,A -85,B 0,C 180,E1 -27977.341,E2 -27977.341} C_VEL
LIN {X 0,Y 73.151,Z 449.779,A -85,B 0,C 180,E1 -27983.103,E2 -27983.103} C_VEL
LIN {X 0,Y 75.613,Z 444.242,A -85,B 0,C 180,E1 -27988.669,E2 -27988.669} C_VEL
LIN {X 0,Y 78.173,Z 438.51,A -85,B 0,C 180,E1 -27993.177,E2 -27993.177} C_VEL
LIN {X 0,Y 81.686,Z 430.391,A -85,B 0,C 180,E1 -27998.037,E2 -27998.037} C_VEL
LIN {X 0,Y 85.044,Z 421.949,A -85,B 0,C 180,E1 -28001.802,E2 -28001.802} C_VEL
LIN {X 0,Y 88.448,Z 412.23,A -85,B 0,C 180,E1 -28004.965,E2 -28004.965} C_VEL
LIN {X 0,Y 91.224,Z 401.823,A -85,B 0,C 180,E1 -28007.369,E2 -28007.369} C_VEL
LIN {X 0,Y 93.173,Z 392.194,A -85,B 0,C 180,E1 -28008.951,E2 -28008.951} C_VEL
LIN {X 0,Y 94.603,Z 382.561,A -85,B 0,C 180,E1 -28009.976,E2 -28009.976} C_VEL
LIN {X 0,Y 96.395,Z 362.165,A -85,B 0,C 180,E1 -28011.379,E2 -28011.379} C_VEL
LIN {X 0,Y 93.026,Z 354.12,A -85,B 0,C 180,E1 -28014.008,E2 -28014.008} C_VEL
LIN {X 0,Y 86.67,Z 342.181,A -85,B 0,C 180,E1 -28019.361,E2 -28019.361} C_VEL
LIN {X 0,Y 81.932,Z 335.013,A -85,B 0,C 180,E1 -28024.065,E2 -28024.065} C_VEL
LIN {X 0,Y 79.421,Z 331.317,A -85,B 0,C 180,E1 -28026.925,E2 -28026.925} C_VEL
LIN {X 0,Y 77.109,Z 328.533,A -85,B 0,C 180,E1 -28029.809,E2 -28029.809} C_VEL
LIN {X 0,Y 76.175,Z 326.704,A -85,B 0,C 180,E1 -28031.225,E2 -28031.225} C_VEL
LIN {X 0,Y 73.685,Z 324.587,A -85,B 0,C 180,E1 -28034.872,E2 -28034.872} C_VEL
LIN {X 0,Y 72.398,Z 322.116,A -85,B 0,C 180,E1 -28037.334,E2 -28037.334} C_VEL
LIN {X 0,Y 72.259,Z 321.297,A -85,B 0,C 180,E1 -28037.933,E2 -28037.933} C_VEL
LIN {X 0,Y 72.309,Z 321.255,A -85,B 0,C 180,E1 -28044.326,E2 -28044.326} C_VEL
LIN {X 0,Y 72.391,Z 321.279,A -85,B 0,C 180,E1 -28050.959,E2 -28050.959} C_VEL
LIN {X 0,Y 72.391,Z 321.243,A -85,B 0,C 180,E1 -28057.148,E2 -28057.148} C_VEL
LIN {X 0,Y 72.72,Z 321.233,A -85,B 0,C 180,E1 -28065.11,E2 -28065.11} C_VEL
LIN {X 0,Y 72.856,Z 321.218,A -85,B 0,C 180,E1 -28068.876,E2 -28068.876} C_VEL
LIN {X 0,Y 73.565,Z 321.123,A -85,B 0,C 180,E1 -28079.999,E2 -28079.999} C_VEL
LIN {X 0,Y 72.856,Z 321.192,A -85,B 0,C 180,E1 -28091.123,E2 -28091.123} C_VEL
LIN {X 0,Y 72.764,Z 321.39,A -85,B 0,C 180,E1 -28094.651,E2 -28094.651} C_VEL
LIN {X 0,Y 73.495,Z 323.877,A -85,B 0,C 180,E1 -28096.306,E2 -28096.306} C_VEL
LIN {X 0,Y 75.224,Z 326.032,A -85,B 0,C 180,E1 -28099.086,E2 -28099.086} C_VEL
LIN {X 0,Y 76.53,Z 326.972,A -85,B 0,C 180,E1 -28100.845,E2 -28100.845} C_VEL
LIN {X 0,Y 78.382,Z 330.212,A -85,B 0,C 180,E1 -28103.445,E2 -28103.445} C_VEL
LIN {X 0,Y 80.008,Z 332.115,A -85,B 0,C 180,E1 -28105.354,E2 -28105.354} C_VEL
LIN {X 0,Y 83.402,Z 337.315,A -85,B 0,C 180,E1 -28109.113,E2 -28109.113} C_VEL
LIN {X 0,Y 87.449,Z 344.111,A -85,B 0,C 180,E1 -28113.023,E2 -28113.023} C_VEL
LIN {X 0,Y 91.677,Z 352.239,A -85,B 0,C 180,E1 -28116.62,E2 -28116.62} C_VEL
LIN {X 0,Y 93.75,Z 357.192,A -85,B 0,C 180,E1 -28118.332,E2 -28118.332} C_VEL
LIN {X 0,Y 95.545,Z 363.439,A -85,B 0,C 180,E1 -28119.938,E2 -28119.938} C_VEL
LIN {X 0,Y 95.804,Z 371.764,A -85,B 0,C 180,E1 -28120.943,E2 -28120.943} C_VEL
LIN {X 0,Y 94.073,Z 389.839,A -85,B 0,C 180,E1 -28122.25,E2 -28122.25} C_VEL
LIN {X 0,Y 91.819,Z 401.894,A -85,B 0,C 180,E1 -28123.767,E2 -28123.767} C_VEL
LIN {X 0,Y 89.25,Z 411.631,A -85,B 0,C 180,E1 -28125.666,E2 -28125.666} C_VEL
LIN {X 0,Y 87.271,Z 418.674,A -85,B 0,C 180,E1 -28127.59,E2 -28127.59} C_VEL
LIN {X 0,Y 84.079,Z 427.03,A -85,B 0,C 180,E1 -28130.406,E2 -28130.406} C_VEL
LIN {X 0,Y 80.971,Z 435.039,A -85,B 0,C 180,E1 -28134.136,E2 -28134.136} C_VEL
LIN {X 0,Y 77.666,Z 442.471,A -85,B 0,C 180,E1 -28138.647,E2 -28138.647} C_VEL
LIN {X 0,Y 74.344,Z 450.021,A -85,B 0,C 180,E1 -28144.825,E2 -28144.825} C_VEL
LIN {X 0,Y 71.519,Z 456.902,A -85,B 0,C 180,E1 -28152.855,E2 -28152.855} C_VEL
LIN {X 0,Y 70.053,Z 462.086,A -85,B 0,C 180,E1 -28161.345,E2 -28161.345} C_VEL
LIN {X 0,Y 69.774,Z 464.713,A -85,B 0,C 180,E1 -28167.113,E2 -28167.113} C_VEL
LIN {X 0,Y 69.823,Z 465.849,A -85,B 0,C 180,E1 -28170,E2 -28170} C_VEL
LIN {X 0,Y 69.825,Z 467.518,A -85,B 0,C 180,E1 -28175.776,E2 -28175.776} C_VEL
LIN {X 0,Y 70.351,Z 468.708,A -85,B 0,C 180,E1 -28181.525,E2 -28181.525} C_VEL
LIN {X 0,Y 71.52,Z 469.457,A -85,B 0,C 180,E1 -28187.145,E2 -28187.145} C_VEL
LIN {X 0,Y 73.386,Z 469.71,A -85,B 0,C 180,E1 -28192.523,E2 -28192.523} C_VEL
LIN {X 0,Y 75.812,Z 469.41,A -85,B 0,C 180,E1 -28197.613,E2 -28197.613} C_VEL
LIN {X 0,Y 78.788,Z 468.683,A -85,B 0,C 180,E1 -28202.357,E2 -28202.357} C_VEL
LIN {X 0,Y 82.37,Z 467.52,A -85,B 0,C 180,E1 -28206.672,E2 -28206.672} C_VEL
LIN {X 0,Y 88.605,Z 464.739,A -85,B 0,C 180,E1 -28212.39,E2 -28212.39} C_VEL
LIN {X 0,Y 95.654,Z 460.764,A -85,B 0,C 180,E1 -28217.282,E2 -28217.282} C_VEL
LIN {X 0,Y 100.634,Z 457.363,A -85,B 0,C 180,E1 -28220.191,E2 -28220.191} C_VEL
LIN {X 0,Y 105.921,Z 453.281,A -85,B 0,C 180,E1 -28222.768,E2 -28222.768} C_VEL
LIN {X 0,Y 111.431,Z 448.406,A -85,B 0,C 180,E1 -28225.074,E2 -28225.074} C_VEL
LIN {X 0,Y 117.133,Z 442.564,A -85,B 0,C 180,E1 -28227.137,E2 -28227.137} C_VEL
LIN {X 0,Y 123.003,Z 435.493,A -85,B 0,C 180,E1 -28228.984,E2 -28228.984} C_VEL
LIN {X 0,Y 128.248,Z 427.998,A -85,B 0,C 180,E1 -28230.449,E2 -28230.449} C_VEL
LIN {X 0,Y 133.632,Z 418.704,A -85,B 0,C 180,E1 -28231.75,E2 -28231.75} C_VEL
LIN {X 0,Y 138.217,Z 408.753,A -85,B 0,C 180,E1 -28232.746,E2 -28232.746} C_VEL
LIN {X 0,Y 141.414,Z 399.551,A -85,B 0,C 180,E1 -28233.449,E2 -28233.449} C_VEL
LIN {X 0,Y 141.495,Z 397.469,A -85,B 0,C 180,E1 -28234.377,E2 -28234.377} C_VEL
LIN {X 0,Y 140.767,Z 394.744,A -85,B 0,C 180,E1 -28237.237,E2 -28237.237} C_VEL
LIN {X 0,Y 140.345,Z 392.984,A -85,B 0,C 180,E1 -28239.48,E2 -28239.48} C_VEL
LIN {X 0,Y 139.747,Z 391.003,A -85,B 0,C 180,E1 -28245.437,E2 -28245.437} C_VEL
LIN {X 0,Y 139.83,Z 391.155,A -85,B 0,C 180,E1 -28248.838,E2 -28248.838} C_VEL
LIN {X 0,Y 140.449,Z 393.033,A -85,B 0,C 180,E1 -28253.739,E2 -28253.739} C_VEL
LIN {X 0,Y 141.311,Z 396.522,A -85,B 0,C 180,E1 -28257.722,E2 -28257.722} C_VEL
LIN {X 0,Y 141.521,Z 397.942,A -85,B 0,C 180,E1 -28258.908,E2 -28258.908} C_VEL
LIN {X 0,Y 138.022,Z 407.936,A -85,B 0,C 180,E1 -28259.86,E2 -28259.86} C_VEL
LIN {X 0,Y 134.125,Z 416.475,A -85,B 0,C 180,E1 -28260.849,E2 -28260.849} C_VEL
LIN {X 0,Y 129.228,Z 425.119,A -85,B 0,C 180,E1 -28262.17,E2 -28262.17} C_VEL
LIN {X 0,Y 124.06,Z 432.644,A -85,B 0,C 180,E1 -28263.693,E2 -28263.693} C_VEL
LIN {X 0,Y 122.79,Z 434.37,A -85,B 0,C 180,E1 -28264.099,E2 -28264.099} C_VEL
LIN {X 0,Y 119.137,Z 438.687,A -85,B 0,C 180,E1 -28264.931,E2 -28264.931} C_VEL
LIN {X 0,Y 111.903,Z 445.252,A -85,B 0,C 180,E1 -28265.813,E2 -28265.813} C_VEL
LIN {X 0,Y 104.141,Z 450.969,A -85,B 0,C 180,E1 -28267.018,E2 -28267.018} C_VEL
LIN {X 0,Y 99.724,Z 453.948,A -85,B 0,C 180,E1 -28268.446,E2 -28268.446} C_VEL
LIN {X 0,Y 93.298,Z 458.049,A -85,B 0,C 180,E1 -28271.695,E2 -28271.695} C_VEL
LIN {X 0,Y 87.414,Z 461.162,A -85,B 0,C 180,E1 -28275.258,E2 -28275.258} C_VEL
LIN {X 0,Y 80.83,Z 463.917,A -85,B 0,C 180,E1 -28280.353,E2 -28280.353} C_VEL
LIN {X 0,Y 76.973,Z 465.208,A -85,B 0,C 180,E1 -28284.074,E2 -28284.074} C_VEL
LIN {X 0,Y 72.541,Z 466.211,A -85,B 0,C 180,E1 -28289.318,E2 -28289.318} C_VEL
LIN {X 0,Y 68.79,Z 466.538,A -85,B 0,C 180,E1 -28295.184,E2 -28295.184} C_VEL
LIN {X 0,Y 65.822,Z 466.205,A -85,B 0,C 180,E1 -28301.636,E2 -28301.636} C_VEL
LIN {X 0,Y 63.151,Z 464.805,A -85,B 0,C 180,E1 -28311.172,E2 -28311.172} C_VEL
LIN {X 0,Y 62.18,Z 462.688,A -85,B 0,C 180,E1 -28319.429,E2 -28319.429} C_VEL
LIN {X 0,Y 62.472,Z 459.775,A -85,B 0,C 180,E1 -28327.516,E2 -28327.516} C_VEL
LIN {X 0,Y 64.1,Z 454.734,A -85,B 0,C 180,E1 -28337.334,E2 -28337.334} C_VEL
LIN {X 0,Y 66.055,Z 450.218,A -85,B 0,C 180,E1 -28343.893,E2 -28343.893} C_VEL
LIN {X 0,Y 68.628,Z 444.745,A -85,B 0,C 180,E1 -28350,E2 -28350} C_VEL
LIN {X 0,Y 71.091,Z 439.703,A -85,B 0,C 180,E1 -28354.427,E2 -28354.427} C_VEL
LIN {X 0,Y 74.655,Z 432.122,A -85,B 0,C 180,E1 -28359.482,E2 -28359.482} C_VEL
LIN {X 0,Y 77.75,Z 425.045,A -85,B 0,C 180,E1 -28363.06,E2 -28363.06} C_VEL
LIN {X 0,Y 81.114,Z 416.394,A -85,B 0,C 180,E1 -28366.355,E2 -28366.355} C_VEL
LIN {X 0,Y 84.063,Z 407.358,A -85,B 0,C 180,E1 -28368.902,E2 -28368.902} C_VEL
LIN {X 0,Y 86.697,Z 396.852,A -85,B 0,C 180,E1 -28371.082,E2 -28371.082} C_VEL
LIN {X 0,Y 88.793,Z 384.77,A -85,B 0,C 180,E1 -28372.605,E2 -28372.605} C_VEL
LIN {X 0,Y 90.829,Z 364.217,A -85,B 0,C 180,E1 -28374.066,E2 -28374.066} C_VEL
LIN {X 0,Y 88.03,Z 357.499,A -85,B 0,C 180,E1 -28376.51,E2 -28376.51} C_VEL
LIN {X 0,Y 82.383,Z 346.529,A -85,B 0,C 180,E1 -28381.98,E2 -28381.98} C_VEL
LIN {X 0,Y 78.496,Z 340.408,A -85,B 0,C 180,E1 -28386.312,E2 -28386.312} C_VEL
LIN {X 0,Y 76.242,Z 337.015,A -85,B 0,C 180,E1 -28389.214,E2 -28389.214} C_VEL
LIN {X 0,Y 73.842,Z 333.518,A -85,B 0,C 180,E1 -28392.76,E2 -28392.76} C_VEL
LIN {X 0,Y 73.106,Z 332.659,A -85,B 0,C 180,E1 -28393.928,E2 -28393.928} C_VEL
LIN {X 0,Y 70.663,Z 329.73,A -85,B 0,C 180,E1 -28398.242,E2 -28398.242} C_VEL
LIN {X 0,Y 69.901,Z 327.997,A -85,B 0,C 180,E1 -28400.008,E2 -28400.008} C_VEL
LIN {X 0,Y 66.551,Z 325.52,A -85,B 0,C 180,E1 -28408.454,E2 -28408.454} C_VEL
LIN {X 0,Y 65.293,Z 322.456,A -85,B 0,C 180,E1 -28414.497,E2 -28414.497} C_VEL
LIN {X 0,Y 65.27,Z 322.142,A -85,B 0,C 180,E1 -28415.338,E2 -28415.338} C_VEL
LIN {X 0,Y 65.624,Z 322.111,A -85,B 0,C 180,E1 -28424.543,E2 -28424.543} C_VEL
LIN {X 0,Y 65.753,Z 322.107,A -85,B 0,C 180,E1 -28427.656,E2 -28427.656} C_VEL
LIN {X 0,Y 66.488,Z 322.001,A -85,B 0,C 180,E1 -28439.999,E2 -28439.999} C_VEL
LIN {X 0,Y 66.369,Z 322.232,A -85,B 0,C 180,E1 -28441.137,E2 -28441.137} C_VEL
LIN {X 0,Y 66.892,Z 324.602,A -85,B 0,C 180,E1 -28443.764,E2 -28443.764} C_VEL
LIN {X 0,Y 68.647,Z 326.92,A -85,B 0,C 180,E1 -28448.833,E2 -28448.833} C_VEL
LIN {X 0,Y 70.278,Z 328.047,A -85,B 0,C 180,E1 -28452.251,E2 -28452.251} C_VEL
LIN {X 0,Y 71.717,Z 331.042,A -85,B 0,C 180,E1 -28455.314,E2 -28455.314} C_VEL
LIN {X 0,Y 73.951,Z 333.453,A -85,B 0,C 180,E1 -28458.977,E2 -28458.977} C_VEL
LIN {X 0,Y 76.284,Z 336.988,A -85,B 0,C 180,E1 -28462.424,E2 -28462.424} C_VEL
LIN {X 0,Y 80.084,Z 342.966,A -85,B 0,C 180,E1 -28467.14,E2 -28467.14} C_VEL
LIN {X 0,Y 84.279,Z 350.447,A -85,B 0,C 180,E1 -28471.636,E2 -28471.636} C_VEL
LIN {X 0,Y 88.534,Z 359.631,A -85,B 0,C 180,E1 -28475.653,E2 -28475.653} C_VEL
LIN {X 0,Y 90.173,Z 366.071,A -85,B 0,C 180,E1 -28477.372,E2 -28477.372} C_VEL
LIN {X 0,Y 90.333,Z 372.143,A -85,B 0,C 180,E1 -28478.159,E2 -28478.159} C_VEL
LIN {X 0,Y 88.465,Z 390.397,A -85,B 0,C 180,E1 -28479.524,E2 -28479.524} C_VEL
LIN {X 0,Y 86.159,Z 401.808,A -85,B 0,C 180,E1 -28481.023,E2 -28481.023} C_VEL
LIN {X 0,Y 83.737,Z 410.61,A -85,B 0,C 180,E1 -28482.747,E2 -28482.747} C_VEL
LIN {X 0,Y 81.038,Z 419.294,A -85,B 0,C 180,E1 -28485.201,E2 -28485.201} C_VEL
LIN {X 0,Y 77.683,Z 427.493,A -85,B 0,C 180,E1 -28488.149,E2 -28488.149} C_VEL
LIN {X 0,Y 74.365,Z 435.382,A -85,B 0,C 180,E1 -28492.101,E2 -28492.101} C_VEL
LIN {X 0,Y 70.864,Z 442.718,A -85,B 0,C 180,E1 -28496.945,E2 -28496.945} C_VEL
LIN {X 0,Y 67.356,Z 450.174,A -85,B 0,C 180,E1 -28503.676,E2 -28503.676} C_VEL
LIN {X 0,Y 64.758,Z 455.98,A -85,B 0,C 180,E1 -28511,E2 -28511} C_VEL
LIN {X 0,Y 63.462,Z 459.773,A -85,B 0,C 180,E1 -28517.204,E2 -28517.204} C_VEL
LIN {X 0,Y 62.699,Z 464.071,A -85,B 0,C 180,E1 -28526.787,E2 -28526.787} C_VEL
LIN {X 0,Y 62.753,Z 465.207,A -85,B 0,C 180,E1 -28530,E2 -28530} C_VEL
LIN {X 0,Y 62.783,Z 467.008,A -85,B 0,C 180,E1 -28536.427,E2 -28536.427} C_VEL
LIN {X 0,Y 63.414,Z 468.324,A -85,B 0,C 180,E1 -28542.806,E2 -28542.806} C_VEL
LIN {X 0,Y 64.768,Z 469.176,A -85,B 0,C 180,E1 -28548.997,E2 -28548.997} C_VEL
LIN {X 0,Y 66.863,Z 469.453,A -85,B 0,C 180,E1 -28554.862,E2 -28554.862} C_VEL
LIN {X 0,Y 69.576,Z 469.274,A -85,B 0,C 180,E1 -28560.334,E2 -28560.334} C_VEL
LIN {X 0,Y 72.877,Z 468.676,A -85,B 0,C 180,E1 -28565.352,E2 -28565.352} C_VEL
LIN {X 0,Y 76.804,Z 467.635,A -85,B 0,C 180,E1 -28569.831,E2 -28569.831} C_VEL
LIN {X 0,Y 83.509,Z 465.018,A -85,B 0,C 180,E1 -28575.67,E2 -28575.67} C_VEL
LIN {X 0,Y 90.995,Z 461.197,A -85,B 0,C 180,E1 -28580.563,E2 -28580.563} C_VEL
LIN {X 0,Y 96.258,Z 457.958,A -85,B 0,C 180,E1 -28583.427,E2 -28583.427} C_VEL
LIN {X 0,Y 103.254,Z 452.886,A -85,B 0,C 180,E1 -28586.488,E2 -28586.488} C_VEL
LIN {X 0,Y 109.011,Z 447.977,A -85,B 0,C 180,E1 -28588.672,E2 -28588.672} C_VEL
LIN {X 0,Y 114.688,Z 442.427,A -85,B 0,C 180,E1 -28590.469,E2 -28590.469} C_VEL
LIN {X 0,Y 121.071,Z 434.999,A -85,B 0,C 180,E1 -28592.277,E2 -28592.277} C_VEL
LIN {X 0,Y 125.726,Z 428.671,A -85,B 0,C 180,E1 -28593.426,E2 -28593.426} C_VEL
LIN {X 0,Y 130.595,Z 420.807,A -85,B 0,C 180,E1 -28594.5,E2 -28594.5} C_VEL
LIN {X 0,Y 135.165,Z 411.747,A -85,B 0,C 180,E1 -28595.374,E2 -28595.374} C_VEL
LIN {X 0,Y 138.639,Z 402.897,A -85,B 0,C 180,E1 -28596.075,E2 -28596.075} C_VEL
LIN {X 0,Y 138.258,Z 400.315,A -85,B 0,C 180,E1 -28599.156,E2 -28599.156} C_VEL
LIN {X 0,Y 137.841,Z 397.839,A -85,B 0,C 180,E1 -28605.628,E2 -28605.628} C_VEL
LIN {X 0,Y 137.908,Z 397.827,A -85,B 0,C 180,E1 -28608.238,E2 -28608.238} C_VEL
LIN {X 0,Y 138.01,Z 398.84,A -85,B 0,C 180,E1 -28611.213,E2 -28611.213} C_VEL
LIN {X 0,Y 138.258,Z 400.451,A -85,B 0,C 180,E1 -28614.165,E2 -28614.165} C_VEL
LIN {X 0,Y 138.499,Z 401.791,A -85,B 0,C 180,E1 -28615.954,E2 -28615.954} C_VEL
LIN {X 0,Y 138.33,Z 402.937,A -85,B 0,C 180,E1 -28616.519,E2 -28616.519} C_VEL
LIN {X 0,Y 134.423,Z 412.492,A -85,B 0,C 180,E1 -28617.397,E2 -28617.397} C_VEL
LIN {X 0,Y 129.171,Z 422.361,A -85,B 0,C 180,E1 -28618.655,E2 -28618.655} C_VEL
LIN {X 0,Y 122.996,Z 431.376,A -85,B 0,C 180,E1 -28620.204,E2 -28620.204} C_VEL
LIN {X 0,Y 117.768,Z 437.791,A -85,B 0,C 180,E1 -28621.711,E2 -28621.711} C_VEL
LIN {X 0,Y 112.031,Z 443.806,A -85,B 0,C 180,E1 -28623.597,E2 -28623.597} C_VEL
LIN {X 0,Y 105.963,Z 449.221,A -85,B 0,C 180,E1 -28625.821,E2 -28625.821} C_VEL
LIN {X 0,Y 99.724,Z 453.948,A -85,B 0,C 180,E1 -28628.446,E2 -28628.446} C_VEL
LIN {X 0,Y 95.228,Z 456.786,A -85,B 0,C 180,E1 -28630.078,E2 -28630.078} C_VEL
LIN {X 0,Y 83.423,Z 462.032,A -85,B 0,C 180,E1 -28633.357,E2 -28633.357} C_VEL
LIN {X 0,Y 76.927,Z 464.12,A -85,B 0,C 180,E1 -28636.127,E2 -28636.127} C_VEL
LIN {X 0,Y 74.153,Z 464.953,A -85,B 0,C 180,E1 -28638.105,E2 -28638.105} C_VEL
LIN {X 0,Y 67.989,Z 466.345,A -85,B 0,C 180,E1 -28644.424,E2 -28644.424} C_VEL
LIN {X 0,Y 64.404,Z 466.658,A -85,B 0,C 180,E1 -28649.196,E2 -28649.196} C_VEL
LIN {X 0,Y 60.692,Z 466.535,A -85,B 0,C 180,E1 -28655.85,E2 -28655.85} C_VEL
LIN {X 0,Y 56.516,Z 465.034,A -85,B 0,C 180,E1 -28668.257,E2 -28668.257} C_VEL
LIN {X 0,Y 55.106,Z 462.387,A -85,B 0,C 180,E1 -28679.328,E2 -28679.328} C_VEL
LIN {X 0,Y 55.355,Z 459.664,A -85,B 0,C 180,E1 -28687.612,E2 -28687.612} C_VEL
LIN {X 0,Y 56.474,Z 456.194,A -85,B 0,C 180,E1 -28695.589,E2 -28695.589} C_VEL
LIN {X 0,Y 58.938,Z 450.665,A -85,B 0,C 180,E1 -28704.869,E2 -28704.869} C_VEL
LIN {X 0,Y 61.599,Z 445.434,A -85,B 0,C 180,E1 -28711.425,E2 -28711.425} C_VEL
LIN {X 0,Y 65.149,Z 438.631,A -85,B 0,C 180,E1 -28717.75,E2 -28717.75} C_VEL
LIN {X 0,Y 68.709,Z 431.624,A -85,B 0,C 180,E1 -28722.554,E2 -28722.554} C_VEL
LIN {X 0,Y 72.052,Z 424.411,A -85,B 0,C 180,E1 -28726.285,E2 -28726.285} C_VEL
LIN {X 0,Y 75.439,Z 416.213,A -85,B 0,C 180,E1 -28729.454,E2 -28729.454} C_VEL
LIN {X 0,Y 79.012,Z 405.721,A -85,B 0,C 180,E1 -28732.416,E2 -28732.416} C_VEL
LIN {X 0,Y 81.897,Z 393.934,A -85,B 0,C 180,E1 -28734.624,E2 -28734.624} C_VEL
LIN {X 0,Y 83.501,Z 384.599,A -85,B 0,C 180,E1 -28735.746,E2 -28735.746} C_VEL
LIN {X 0,Y 85.405,Z 366.045,A -85,B 0,C 180,E1 -28737.115,E2 -28737.115} C_VEL
LIN {X 0,Y 82.151,Z 358.655,A -85,B 0,C 180,E1 -28740.419,E2 -28740.419} C_VEL
LIN {X 0,Y 78.008,Z 350.376,A -85,B 0,C 180,E1 -28745.141,E2 -28745.141} C_VEL
LIN {X 0,Y 73.397,Z 342.891,A -85,B 0,C 180,E1 -28751.411,E2 -28751.411} C_VEL
LIN {X 0,Y 70.726,Z 338.903,A -85,B 0,C 180,E1 -28755.925,E2 -28755.925} C_VEL
LIN {X 0,Y 68.221,Z 335.469,A -85,B 0,C 180,E1 -28761.055,E2 -28761.055} C_VEL
LIN {X 0,Y 67.691,Z 334.504,A -85,B 0,C 180,E1 -28762.412,E2 -28762.412} C_VEL
LIN {X 0,Y 64.911,Z 331.9,A -85,B 0,C 180,E1 -28770.781,E2 -28770.781} C_VEL
LIN {X 0,Y 63.966,Z 329.127,A -85,B 0,C 180,E1 -28776.528,E2 -28776.528} C_VEL
LIN {X 0,Y 63.259,Z 328.743,A -85,B 0,C 180,E1 -28787.161,E2 -28787.161} C_VEL
LIN {X 0,Y 64.775,Z 329.082,A -85,B 0,C 180,E1 -28798.834,E2 -28798.834} C_VEL
LIN {X 0,Y 65.525,Z 331.64,A -85,B 0,C 180,E1 -28802.689,E2 -28802.689} C_VEL
LIN {X 0,Y 67.345,Z 333.891,A -85,B 0,C 180,E1 -28808.249,E2 -28808.249} C_VEL
LIN {X 0,Y 68.168,Z 334.699,A -85,B 0,C 180,E1 -28810.206,E2 -28810.206} C_VEL
LIN {X 0,Y 70.01,Z 338.007,A -85,B 0,C 180,E1 -28814.336,E2 -28814.336} C_VEL
LIN {X 0,Y 71.457,Z 339.757,A -85,B 0,C 180,E1 -28816.936,E2 -28816.936} C_VEL
LIN {X 0,Y 74.475,Z 344.706,A -85,B 0,C 180,E1 -28821.831,E2 -28821.831} C_VEL
LIN {X 0,Y 77.397,Z 349.521,A -85,B 0,C 180,E1 -28825.731,E2 -28825.731} C_VEL
LIN {X 0,Y 81.807,Z 358.4,A -85,B 0,C 180,E1 -28830.885,E2 -28830.885} C_VEL
LIN {X 0,Y 84.09,Z 364.126,A -85,B 0,C 180,E1 -28833.345,E2 -28833.345} C_VEL
LIN {X 0,Y 85.012,Z 368.421,A -85,B 0,C 180,E1 -28834.529,E2 -28834.529} C_VEL
LIN {X 0,Y 84.965,Z 373.191,A -85,B 0,C 180,E1 -28835.11,E2 -28835.11} C_VEL
LIN {X 0,Y 83.02,Z 390.83,A -85,B 0,C 180,E1 -28836.476,E2 -28836.476} C_VEL
LIN {X 0,Y 80.893,Z 400.896,A -85,B 0,C 180,E1 -28837.801,E2 -28837.801} C_VEL
LIN {X 0,Y 77.873,Z 411.277,A -85,B 0,C 180,E1 -28839.906,E2 -28839.906} C_VEL
LIN {X 0,Y 74.966,Z 419.774,A -85,B 0,C 180,E1 -28842.417,E2 -28842.417} C_VEL
LIN {X 0,Y 71.435,Z 427.859,A -85,B 0,C 180,E1 -28845.496,E2 -28845.496} C_VEL
LIN {X 0,Y 67.878,Z 435.65,A -85,B 0,C 180,E1 -28849.677,E2 -28849.677} C_VEL
LIN {X 0,Y 63.282,Z 444.575,A -85,B 0,C 180,E1 -28856.27,E2 -28856.27} C_VEL
LIN {X 0,Y 59.749,Z 451.476,A -85,B 0,C 180,E1 -28863.827,E2 -28863.827} C_VEL
LIN {X 0,Y 57.241,Z 456.961,A -85,B 0,C 180,E1 -28872.125,E2 -28872.125} C_VEL
LIN {X 0,Y 56.077,Z 460.523,A -85,B 0,C 180,E1 -28879.165,E2 -28879.165} C_VEL
LIN {X 0,Y 55.641,Z 463.43,A -85,B 0,C 180,E1 -28886.379,E2 -28886.379} C_VEL
LIN {X 0,Y 55.666,Z 464.565,A -85,B 0,C 180,E1 -28890,E2 -28890} C_VEL
LIN {X 0,Y 55.747,Z 466.498,A -85,B 0,C 180,E1 -28897.242,E2 -28897.242} C_VEL
LIN {X 0,Y 56.526,Z 467.939,A -85,B 0,C 180,E1 -28904.398,E2 -28904.398} C_VEL
LIN {X 0,Y 58.105,Z 468.817,A -85,B 0,C 180,E1 -28911.275,E2 -28911.275} C_VEL
LIN {X 0,Y 60.479,Z 469.19,A -85,B 0,C 180,E1 -28917.697,E2 -28917.697} C_VEL
LIN {X 0,Y 63.528,Z 469.143,A -85,B 0,C 180,E1 -28923.582,E2 -28923.582} C_VEL
LIN {X 0,Y 67.204,Z 468.679,A -85,B 0,C 180,E1 -28928.861,E2 -28928.861} C_VEL
LIN {X 0,Y 71.488,Z 467.681,A -85,B 0,C 180,E1 -28933.484,E2 -28933.484} C_VEL
LIN {X 0,Y 78.724,Z 465.286,A -85,B 0,C 180,E1 -28939.359,E2 -28939.359} C_VEL
LIN {X 0,Y 86.666,Z 461.63,A -85,B 0,C 180,E1 -28944.184,E2 -28944.184} C_VEL
LIN {X 0,Y 92.219,Z 458.558,A -85,B 0,C 180,E1 -28946.959,E2 -28946.959} C_VEL
LIN {X 0,Y 99.53,Z 453.697,A -85,B 0,C 180,E1 -28949.878,E2 -28949.878} C_VEL
LIN {X 0,Y 107.039,Z 447.626,A -85,B 0,C 180,E1 -28952.419,E2 -28952.419} C_VEL
LIN {X 0,Y 112.934,Z 442.089,A -85,B 0,C 180,E1 -28953.997,E2 -28953.997} C_VEL
LIN {X 0,Y 119.565,Z 434.588,A -85,B 0,C 180,E1 -28955.652,E2 -28955.652} C_VEL
LIN {X 0,Y 125.086,Z 427.145,A -85,B 0,C 180,E1 -28956.803,E2 -28956.803} C_VEL
LIN {X 0,Y 130.194,Z 418.834,A -85,B 0,C 180,E1 -28957.731,E2 -28957.731} C_VEL
LIN {X 0,Y 134.785,Z 409.517,A -85,B 0,C 180,E1 -28958.513,E2 -28958.513} C_VEL
LIN {X 0,Y 135.671,Z 407.471,A -85,B 0,C 180,E1 -28958.74,E2 -28958.74} C_VEL
LIN {X 0,Y 135.416,Z 405.856,A -85,B 0,C 180,E1 -28961.857,E2 -28961.857} C_VEL
LIN {X 0,Y 135.358,Z 404.764,A -85,B 0,C 180,E1 -28964.954,E2 -28964.954} C_VEL
LIN {X 0,Y 135.442,Z 404.492,A -85,B 0,C 180,E1 -28968.021,E2 -28968.021} C_VEL
LIN {X 0,Y 135.47,Z 405.544,A -85,B 0,C 180,E1 -28971.047,E2 -28971.047} C_VEL
LIN {X 0,Y 135.528,Z 406.71,A -85,B 0,C 180,E1 -28973.3,E2 -28973.3} C_VEL
LIN {X 0,Y 134.976,Z 408.368,A -85,B 0,C 180,E1 -28974.023,E2 -28974.023} C_VEL
LIN {X 0,Y 130.528,Z 417.478,A -85,B 0,C 180,E1 -28974.914,E2 -28974.914} C_VEL
LIN {X 0,Y 125.52,Z 425.709,A -85,B 0,C 180,E1 -28975.983,E2 -28975.983} C_VEL
LIN {X 0,Y 119.6,Z 433.682,A -85,B 0,C 180,E1 -28977.346,E2 -28977.346} C_VEL
LIN {X 0,Y 112.453,Z 441.64,A -85,B 0,C 180,E1 -28979.285,E2 -28979.285} C_VEL
LIN {X 0,Y 103.724,Z 449.298,A -85,B 0,C 180,E1 -28982.026,E2 -28982.026} C_VEL
LIN {X 0,Y 95.966,Z 454.807,A -85,B 0,C 180,E1 -28984.962,E2 -28984.962} C_VEL
LIN {X 0,Y 89.134,Z 458.795,A -85,B 0,C 180,E1 -28988.117,E2 -28988.117} C_VEL
LIN {X 0,Y 82.564,Z 461.909,A -85,B 0,C 180,E1 -28991.799,E2 -28991.799} C_VEL
LIN {X 0,Y 76.727,Z 464.119,A -85,B 0,C 180,E1 -28995.95,E2 -28995.95} C_VEL
LIN {X 0,Y 74.153,Z 464.953,A -85,B 0,C 180,E1 -28998.105,E2 -28998.105} C_VEL
LIN {X 0,Y 69.95,Z 466.013,A -85,B 0,C 180,E1 -29001.307,E2 -29001.307} C_VEL
LIN {X 0,Y 62.09,Z 466.896,A -85,B 0,C 180,E1 -29006.525,E2 -29006.525} C_VEL
LIN {X 0,Y 54.831,Z 466.701,A -85,B 0,C 180,E1 -29013.194,E2 -29013.194} C_VEL
LIN {X 0,Y 51.827,Z 466.051,A -85,B 0,C 180,E1 -29018.64,E2 -29018.64} C_VEL
LIN {X 0,Y 49.907,Z 465.143,A -85,B 0,C 180,E1 -29025.245,E2 -29025.245} C_VEL
LIN {X 0,Y 48.331,Z 463.28,A -85,B 0,C 180,E1 -29034.435,E2 -29034.435} C_VEL
LIN {X 0,Y 48.335,Z 459.139,A -85,B 0,C 180,E1 -29048.685,E2 -29048.685} C_VEL
LIN {X 0,Y 50.036,Z 454.651,A -85,B 0,C 180,E1 -29059.495,E2 -29059.495} C_VEL
LIN {X 0,Y 52.542,Z 449.783,A -85,B 0,C 180,E1 -29068.084,E2 -29068.084} C_VEL
LIN {X 0,Y 55.821,Z 443.986,A -85,B 0,C 180,E1 -29075.601,E2 -29075.601} C_VEL
LIN {X 0,Y 59.605,Z 437.304,A -85,B 0,C 180,E1 -29081.908,E2 -29081.908} C_VEL
LIN {X 0,Y 64.14,Z 428.922,A -85,B 0,C 180,E1 -29087.537,E2 -29087.537} C_VEL
LIN {X 0,Y 68.866,Z 418.795,A -85,B 0,C 180,E1 -29092.091,E2 -29092.091} C_VEL
LIN {X 0,Y 71.904,Z 411.156,A -85,B 0,C 180,E1 -29094.544,E2 -29094.544} C_VEL
LIN {X 0,Y 74.922,Z 401.539,A -85,B 0,C 180,E1 -29096.835,E2 -29096.835} C_VEL
LIN {X 0,Y 77.154,Z 392.13,A -85,B 0,C 180,E1 -29098.418,E2 -29098.418} C_VEL
LIN {X 0,Y 78.77,Z 382.591,A -85,B 0,C 180,E1 -29099.442,E2 -29099.442} C_VEL
LIN {X 0,Y 80.31,Z 368.259,A -85,B 0,C 180,E1 -29100.468,E2 -29100.468} C_VEL
LIN {X 0,Y 75.654,Z 357.843,A -85,B 0,C 180,E1 -29106.152,E2 -29106.152} C_VEL
LIN {X 0,Y 72.311,Z 351.623,A -85,B 0,C 180,E1 -29110.999,E2 -29110.999} C_VEL
LIN {X 0,Y 70.304,Z 348.245,A -85,B 0,C 180,E1 -29114.406,E2 -29114.406} C_VEL
LIN {X 0,Y 68.302,Z 345.04,A -85,B 0,C 180,E1 -29118.276,E2 -29118.276} C_VEL
LIN {X 0,Y 65.794,Z 341.095,A -85,B 0,C 180,E1 -29124.49,E2 -29124.49} C_VEL
LIN {X 0,Y 63.429,Z 338.445,A -85,B 0,C 180,E1 -29132.847,E2 -29132.847} C_VEL
LIN {X 0,Y 62.689,Z 336.053,A -85,B 0,C 180,E1 -29138.631,E2 -29138.631} C_VEL
LIN {X 0,Y 62.795,Z 335.861,A -85,B 0,C 180,E1 -29153.573,E2 -29153.573} C_VEL
LIN {X 0,Y 63.377,Z 336.163,A -85,B 0,C 180,E1 -29157.094,E2 -29157.094} C_VEL
LIN {X 0,Y 64.647,Z 339.415,A -85,B 0,C 180,E1 -29163.408,E2 -29163.408} C_VEL
LIN {X 0,Y 66.164,Z 341.196,A -85,B 0,C 180,E1 -29168.013,E2 -29168.013} C_VEL
LIN {X 0,Y 68.26,Z 344.802,A -85,B 0,C 180,E1 -29173.173,E2 -29173.173} C_VEL
LIN {X 0,Y 69.259,Z 346.429,A -85,B 0,C 180,E1 -29175.205,E2 -29175.205} C_VEL
LIN {X 0,Y 71.444,Z 350.196,A -85,B 0,C 180,E1 -29179.204,E2 -29179.204} C_VEL
LIN {X 0,Y 74.308,Z 355.458,A -85,B 0,C 180,E1 -29183.635,E2 -29183.635} C_VEL
LIN {X 0,Y 77.937,Z 363.374,A -85,B 0,C 180,E1 -29188.439,E2 -29188.439} C_VEL
LIN {X 0,Y 79.696,Z 368.243,A -85,B 0,C 180,E1 -29190.651,E2 -29190.651} C_VEL
LIN {X 0,Y 80.04,Z 370.399,A -85,B 0,C 180,E1 -29191.239,E2 -29191.239} C_VEL
LIN {X 0,Y 79.623,Z 376.744,A -85,B 0,C 180,E1 -29191.834,E2 -29191.834} C_VEL
LIN {X 0,Y 77.771,Z 391.637,A -85,B 0,C 180,E1 -29193.073,E2 -29193.073} C_VEL
LIN {X 0,Y 75.186,Z 402.364,A -85,B 0,C 180,E1 -29194.54,E2 -29194.54} C_VEL
LIN {X 0,Y 72.237,Z 411.948,A -85,B 0,C 180,E1 -29196.619,E2 -29196.619} C_VEL
LIN {X 0,Y 69.106,Z 420.255,A -85,B 0,C 180,E1 -29199.156,E2 -29199.156} C_VEL
LIN {X 0,Y 65.383,Z 428.23,A -85,B 0,C 180,E1 -29202.356,E2 -29202.356} C_VEL
LIN {X 0,Y 61.534,Z 435.917,A -85,B 0,C 180,E1 -29206.744,E2 -29206.744} C_VEL
LIN {X 0,Y 56.606,Z 444.726,A -85,B 0,C 180,E1 -29213.862,E2 -29213.862} C_VEL
LIN {X 0,Y 52.756,Z 451.539,A -85,B 0,C 180,E1 -29222.209,E2 -29222.209} C_VEL
LIN {X 0,Y 50.528,Z 456.014,A -85,B 0,C 180,E1 -29229.652,E2 -29229.652} C_VEL
LIN {X 0,Y 49.126,Z 459.725,A -85,B 0,C 180,E1 -29237.609,E2 -29237.609} C_VEL
LIN {X 0,Y 48.569,Z 462.724,A -85,B 0,C 180,E1 -29245.851,E2 -29245.851} C_VEL
LIN {X 0,Y 48.538,Z 465.006,A -85,B 0,C 180,E1 -29254.151,E2 -29254.151} C_VEL
LIN {X 0,Y 49.702,Z 467.481,A -85,B 0,C 180,E1 -29266.427,E2 -29266.427} C_VEL
LIN {X 0,Y 51.564,Z 468.419,A -85,B 0,C 180,E1 -29274.134,E2 -29274.134} C_VEL
LIN {X 0,Y 54.284,Z 468.925,A -85,B 0,C 180,E1 -29281.188,E2 -29281.188} C_VEL
LIN {X 0,Y 57.727,Z 469.013,A -85,B 0,C 180,E1 -29287.496,E2 -29287.496} C_VEL
LIN {X 0,Y 61.833,Z 468.63,A -85,B 0,C 180,E1 -29292.996,E2 -29292.996} C_VEL
LIN {X 0,Y 66.512,Z 467.686,A -85,B 0,C 180,E1 -29297.7,E2 -29297.7} C_VEL
LIN {X 0,Y 71.622,Z 466.299,A -85,B 0,C 180,E1 -29301.719,E2 -29301.719} C_VEL
LIN {X 0,Y 79.878,Z 463.299,A -85,B 0,C 180,E1 -29306.701,E2 -29306.701} C_VEL
LIN {X 0,Y 88.562,Z 459.097,A -85,B 0,C 180,E1 -29310.797,E2 -29310.797} C_VEL
LIN {X 0,Y 97.75,Z 453.377,A -85,B 0,C 180,E1 -29313.986,E2 -29313.986} C_VEL
LIN {X 0,Y 105.761,Z 447.1,A -85,B 0,C 180,E1 -29316.334,E2 -29316.334} C_VEL
LIN {X 0,Y 111.959,Z 441.387,A -85,B 0,C 180,E1 -29317.73,E2 -29317.73} C_VEL
LIN {X 0,Y 118.482,Z 434.185,A -85,B 0,C 180,E1 -29319.101,E2 -29319.101} C_VEL
LIN {X 0,Y 124.254,Z 426.577,A -85,B 0,C 180,E1 -29320.103,E2 -29320.103} C_VEL
LIN {X 0,Y 128.785,Z 419.427,A -85,B 0,C 180,E1 -29320.795,E2 -29320.795} C_VEL
LIN {X 0,Y 132.388,Z 412.619,A -85,B 0,C 180,E1 -29321.427,E2 -29321.427} C_VEL
LIN {X 0,Y 132.425,Z 411.405,A -85,B 0,C 180,E1 -29324.612,E2 -29324.612} C_VEL
LIN {X 0,Y 132.53,Z 410.996,A -85,B 0,C 180,E1 -29327.754,E2 -29327.754} C_VEL
LIN {X 0,Y 132.41,Z 412.18,A -85,B 0,C 180,E1 -29331.223,E2 -29331.223} C_VEL
LIN {X 0,Y 126.786,Z 422.39,A -85,B 0,C 180,E1 -29332.311,E2 -29332.311} C_VEL
LIN {X 0,Y 120.231,Z 431.491,A -85,B 0,C 180,E1 -29333.561,E2 -29333.561} C_VEL
LIN {X 0,Y 114.683,Z 437.903,A -85,B 0,C 180,E1 -29334.748,E2 -29334.748} C_VEL
LIN {X 0,Y 107.746,Z 444.624,A -85,B 0,C 180,E1 -29336.468,E2 -29336.468} C_VEL
LIN {X 0,Y 101.959,Z 449.39,A -85,B 0,C 180,E1 -29338.092,E2 -29338.092} C_VEL
LIN {X 0,Y 93.72,Z 455.003,A -85,B 0,C 180,E1 -29340.798,E2 -29340.798} C_VEL
LIN {X 0,Y 84.134,Z 460.192,A -85,B 0,C 180,E1 -29344.792,E2 -29344.792} C_VEL
LIN {X 0,Y 78.053,Z 462.689,A -85,B 0,C 180,E1 -29347.937,E2 -29347.937} C_VEL
LIN {X 0,Y 71.853,Z 464.712,A -85,B 0,C 180,E1 -29352.02,E2 -29352.02} C_VEL
LIN {X 0,Y 63.485,Z 466.553,A -85,B 0,C 180,E1 -29359.398,E2 -29359.398} C_VEL
LIN {X 0,Y 55.481,Z 466.785,A -85,B 0,C 180,E1 -29370.445,E2 -29370.445} C_VEL
LIN {X 0,Y 51.827,Z 466.051,A -85,B 0,C 180,E1 -29378.64,E2 -29378.64} C_VEL
LIN {X 0,Y 49.35,Z 465.207,A -85,B 0,C 180,E1 -29384.596,E2 -29384.596} C_VEL
LIN {X 0,Y 44.773,Z 462.932,A -85,B 0,C 180,E1 -29394.93,E2 -29394.93} C_VEL
LIN {X 0,Y 41.747,Z 459.677,A -85,B 0,C 180,E1 -29406.814,E2 -29406.814} C_VEL
LIN {X 0,Y 41.829,Z 457.246,A -85,B 0,C 180,E1 -29414.351,E2 -29414.351} C_VEL
LIN {X 0,Y 44.79,Z 451.447,A -85,B 0,C 180,E1 -29427.752,E2 -29427.752} C_VEL
LIN {X 0,Y 48.066,Z 446.095,A -85,B 0,C 180,E1 -29436.296,E2 -29436.296} C_VEL
LIN {X 0,Y 52.296,Z 439.408,A -85,B 0,C 180,E1 -29443.776,E2 -29443.776} C_VEL
LIN {X 0,Y 56.324,Z 432.689,A -85,B 0,C 180,E1 -29449.119,E2 -29449.119} C_VEL
LIN {X 0,Y 60.91,Z 424.221,A -85,B 0,C 180,E1 -29453.871,E2 -29453.871} C_VEL
LIN {X 0,Y 65.032,Z 415.377,A -85,B 0,C 180,E1 -29457.341,E2 -29457.341} C_VEL
LIN {X 0,Y 69.372,Z 403.649,A -85,B 0,C 180,E1 -29460.433,E2 -29460.433} C_VEL
LIN {X 0,Y 72.147,Z 393.069,A -85,B 0,C 180,E1 -29462.262,E2 -29462.262} C_VEL
LIN {X 0,Y 73.946,Z 383.129,A -85,B 0,C 180,E1 -29463.358,E2 -29463.358} C_VEL
LIN {X 0,Y 75.345,Z 370.568,A -85,B 0,C 180,E1 -29464.317,E2 -29464.317} C_VEL
LIN {X 0,Y 71.292,Z 360.863,A -85,B 0,C 180,E1 -29470.395,E2 -29470.395} C_VEL
LIN {X 0,Y 67.964,Z 354.525,A -85,B 0,C 180,E1 -29476.429,E2 -29476.429} C_VEL
LIN {X 0,Y 65.852,Z 350.935,A -85,B 0,C 180,E1 -29481.169,E2 -29481.169} C_VEL
LIN {X 0,Y 63.993,Z 347.639,A -85,B 0,C 180,E1 -29486.692,E2 -29486.692} C_VEL
LIN {X 0,Y 62.041,Z 344.981,A -85,B 0,C 180,E1 -29494.988,E2 -29494.988} C_VEL
LIN {X 0,Y 61.57,Z 343.039,A -85,B 0,C 180,E1 -29499.974,E2 -29499.974} C_VEL
LIN {X 0,Y 62.019,Z 342.924,A -85,B 0,C 180,E1 -29514.894,E2 -29514.894} C_VEL
LIN {X 0,Y 63.597,Z 346.718,A -85,B 0,C 180,E1 -29523.39,E2 -29523.39} C_VEL
LIN {X 0,Y 64.317,Z 347.7,A -85,B 0,C 180,E1 -29525.83,E2 -29525.83} C_VEL
LIN {X 0,Y 66.869,Z 352.493,A -85,B 0,C 180,E1 -29532.792,E2 -29532.792} C_VEL
LIN {X 0,Y 69.638,Z 357.681,A -85,B 0,C 180,E1 -29538.376,E2 -29538.376} C_VEL
LIN {X 0,Y 72.822,Z 364.801,A -85,B 0,C 180,E1 -29543.734,E2 -29543.734} C_VEL
LIN {X 0,Y 75.297,Z 371.66,A -85,B 0,C 180,E1 -29547.408,E2 -29547.408} C_VEL
LIN {X 0,Y 74.883,Z 377.053,A -85,B 0,C 180,E1 -29547.909,E2 -29547.909} C_VEL
LIN {X 0,Y 72.893,Z 391.867,A -85,B 0,C 180,E1 -29549.16,E2 -29549.16} C_VEL
LIN {X 0,Y 70.151,Z 402.538,A -85,B 0,C 180,E1 -29550.595,E2 -29550.595} C_VEL
LIN {X 0,Y 67.503,Z 410.71,A -85,B 0,C 180,E1 -29552.305,E2 -29552.305} C_VEL
LIN {X 0,Y 64.206,Z 419.15,A -85,B 0,C 180,E1 -29554.822,E2 -29554.822} C_VEL
LIN {X 0,Y 60.184,Z 427.259,A -85,B 0,C 180,E1 -29557.982,E2 -29557.982} C_VEL
LIN {X 0,Y 55.999,Z 435.075,A -85,B 0,C 180,E1 -29562.498,E2 -29562.498} C_VEL
LIN {X 0,Y 52.079,Z 441.497,A -85,B 0,C 180,E1 -29567.567,E2 -29567.567} C_VEL
LIN {X 0,Y 48.249,Z 447.637,A -85,B 0,C 180,E1 -29574.364,E2 -29574.364} C_VEL
LIN {X 0,Y 44.504,Z 453.888,A -85,B 0,C 180,E1 -29584.261,E2 -29584.261} C_VEL
LIN {X 0,Y 42.237,Z 458.833,A -85,B 0,C 180,E1 -29595.547,E2 -29595.547} C_VEL
LIN {X 0,Y 41.538,Z 463.232,A -85,B 0,C 180,E1 -29610,E2 -29610} C_VEL
LIN {X 0,Y 41.762,Z 465.408,A -85,B 0,C 180,E1 -29619.688,E2 -29619.688} C_VEL
LIN {X 0,Y 42.94,Z 466.952,A -85,B 0,C 180,E1 -29629.107,E2 -29629.107} C_VEL
LIN {X 0,Y 45.178,Z 468.021,A -85,B 0,C 180,E1 -29637.818,E2 -29637.818} C_VEL
LIN {X 0,Y 48.346,Z 468.66,A -85,B 0,C 180,E1 -29645.553,E2 -29645.553} C_VEL
LIN {X 0,Y 52.257,Z 468.868,A -85,B 0,C 180,E1 -29652.254,E2 -29652.254} C_VEL
LIN {X 0,Y 56.846,Z 468.513,A -85,B 0,C 180,E1 -29657.882,E2 -29657.882} C_VEL
LIN {X 0,Y 61.956,Z 467.704,A -85,B 0,C 180,E1 -29662.563,E2 -29662.563} C_VEL
LIN {X 0,Y 67.466,Z 466.463,A -85,B 0,C 180,E1 -29666.443,E2 -29666.443} C_VEL
LIN {X 0,Y 76.219,Z 463.615,A -85,B 0,C 180,E1 -29671.157,E2 -29671.157} C_VEL
LIN {X 0,Y 85.336,Z 459.576,A -85,B 0,C 180,E1 -29674.944,E2 -29674.944} C_VEL
LIN {X 0,Y 88.553,Z 457.961,A -85,B 0,C 180,E1 -29675.877,E2 -29675.877} C_VEL
LIN {X 0,Y 94.867,Z 454.181,A -85,B 0,C 180,E1 -29677.819,E2 -29677.819} C_VEL
LIN {X 0,Y 104.572,Z 446.991,A -85,B 0,C 180,E1 -29680.199,E2 -29680.199} C_VEL
LIN {X 0,Y 111.187,Z 441.059,A -85,B 0,C 180,E1 -29681.46,E2 -29681.46} C_VEL
LIN {X 0,Y 117.845,Z 433.898,A -85,B 0,C 180,E1 -29682.586,E2 -29682.586} C_VEL
LIN {X 0,Y 123.74,Z 426.267,A -85,B 0,C 180,E1 -29683.418,E2 -29683.418} C_VEL
LIN {X 0,Y 128.081,Z 419.561,A -85,B 0,C 180,E1 -29683.954,E2 -29683.954} C_VEL
LIN {X 0,Y 129.046,Z 417.873,A -85,B 0,C 180,E1 -29684.199,E2 -29684.199} C_VEL
LIN {X 0,Y 129.188,Z 417.334,A -85,B 0,C 180,E1 -29687.432,E2 -29687.432} C_VEL
LIN {X 0,Y 129.035,Z 417.714,A -85,B 0,C 180,E1 -29688.624,E2 -29688.624} C_VEL
LIN {X 0,Y 124.056,Z 425.572,A -85,B 0,C 180,E1 -29689.411,E2 -29689.411} C_VEL
LIN {X 0,Y 118.7,Z 432.577,A -85,B 0,C 180,E1 -29690.283,E2 -29690.283} C_VEL
LIN {X 0,Y 113.794,Z 438.072,A -85,B 0,C 180,E1 -29691.166,E2 -29691.166} C_VEL
LIN {X 0,Y 106.269,Z 445.103,A -85,B 0,C 180,E1 -29692.737,E2 -29692.737} C_VEL
LIN {X 0,Y 98.841,Z 450.826,A -85,B 0,C 180,E1 -29694.52,E2 -29694.52} C_VEL
LIN {X 0,Y 89.713,Z 456.544,A -85,B 0,C 180,E1 -29697.175,E2 -29697.175} C_VEL
LIN {X 0,Y 81.919,Z 460.398,A -85,B 0,C 180,E1 -29700.001,E2 -29700.001} C_VEL
LIN {X 0,Y 73.94,Z 463.47,A -85,B 0,C 180,E1 -29703.631,E2 -29703.631} C_VEL
LIN {X 0,Y 64.184,Z 465.99,A -85,B 0,C 180,E1 -29709.787,E2 -29709.787} C_VEL
LIN {X 0,Y 58.191,Z 466.904,A -85,B 0,C 180,E1 -29714.948,E2 -29714.948} C_VEL
LIN {X 0,Y 52.78,Z 467.173,A -85,B 0,C 180,E1 -29721.242,E2 -29721.242} C_VEL
LIN {X 0,Y 48.137,Z 466.77,A -85,B 0,C 180,E1 -29728.84,E2 -29728.84} C_VEL
LIN {X 0,Y 43.859,Z 465.465,A -85,B 0,C 180,E1 -29739.865,E2 -29739.865} C_VEL
LIN {X 0,Y 41.294,Z 462.998,A -85,B 0,C 180,E1 -29753.44,E2 -29753.44} C_VEL
LIN {X 0,Y 40.962,Z 460.3,A -85,B 0,C 180,E1 -29764.654,E2 -29764.654} C_VEL
LIN {X 0,Y 41.829,Z 457.246,A -85,B 0,C 180,E1 -29774.351,E2 -29774.351} C_VEL
LIN {X 0,Y 42.456,Z 454.645,A -85,B 0,C 180,E1 -29781.506,E2 -29781.506} C_VEL
LIN {X 0,Y 42.649,Z 451.687,A -85,B 0,C 180,E1 -29788.455,E2 -29788.455} C_VEL
LIN {X 0,Y 43.74,Z 444.825,A -85,B 0,C 180,E1 -29801.456,E2 -29801.456} C_VEL
LIN {X 0,Y 45.489,Z 440.929,A -85,B 0,C 180,E1 -29806.794,E2 -29806.794} C_VEL
LIN {X 0,Y 46.328,Z 439.524,A -85,B 0,C 180,E1 -29808.255,E2 -29808.255} C_VEL
LIN {X 0,Y 51.193,Z 432.069,A -85,B 0,C 180,E1 -29814.321,E2 -29814.321} C_VEL
LIN {X 0,Y 55.586,Z 424.561,A -85,B 0,C 180,E1 -29818.51,E2 -29818.51} C_VEL
LIN {X 0,Y 59.911,Z 415.965,A -85,B 0,C 180,E1 -29821.861,E2 -29821.861} C_VEL
LIN {X 0,Y 64.164,Z 405.512,A -85,B 0,C 180,E1 -29824.678,E2 -29824.678} C_VEL
LIN {X 0,Y 67.378,Z 394.285,A -85,B 0,C 180,E1 -29826.674,E2 -29826.674} C_VEL
LIN {X 0,Y 69.357,Z 384.565,A -85,B 0,C 180,E1 -29827.714,E2 -29827.714} C_VEL
LIN {X 0,Y 70.791,Z 373.031,A -85,B 0,C 180,E1 -29828.591,E2 -29828.591} C_VEL
LIN {X 0,Y 67.963,Z 365.691,A -85,B 0,C 180,E1 -29833.794,E2 -29833.794} C_VEL
LIN {X 0,Y 65.233,Z 359.942,A -85,B 0,C 180,E1 -29839.727,E2 -29839.727} C_VEL
LIN {X 0,Y 63.654,Z 356.868,A -85,B 0,C 180,E1 -29844.087,E2 -29844.087} C_VEL
LIN {X 0,Y 62.353,Z 354.242,A -85,B 0,C 180,E1 -29848.746,E2 -29848.746} C_VEL
LIN {X 0,Y 60.738,Z 351.532,A -85,B 0,C 180,E1 -29857.241,E2 -29857.241} C_VEL
LIN {X 0,Y 60.51,Z 350.028,A -85,B 0,C 180,E1 -29861.046,E2 -29861.046} C_VEL
LIN {X 0,Y 60.854,Z 349.972,A -85,B 0,C 180,E1 -29873.665,E2 -29873.665} C_VEL
LIN {X 0,Y 62.128,Z 353.414,A -85,B 0,C 180,E1 -29881.708,E2 -29881.708} C_VEL
LIN {X 0,Y 62.638,Z 354.408,A -85,B 0,C 180,E1 -29883.825,E2 -29883.825} C_VEL
LIN {X 0,Y 64.687,Z 358.729,A -85,B 0,C 180,E1 -29890.425,E2 -29890.425} C_VEL
LIN {X 0,Y 67.172,Z 364.08,A -85,B 0,C 180,E1 -29896.241,E2 -29896.241} C_VEL
LIN {X 0,Y 69.971,Z 371.259,A -85,B 0,C 180,E1 -29901.687,E2 -29901.687} C_VEL
LIN {X 0,Y 70.862,Z 374.004,A -85,B 0,C 180,E1 -29903.28,E2 -29903.28} C_VEL
LIN {X 0,Y 68.76,Z 390.217,A -85,B 0,C 180,E1 -29904.531,E2 -29904.531} C_VEL
LIN {X 0,Y 65.85,Z 401.512,A -85,B 0,C 180,E1 -29905.891,E2 -29905.891} C_VEL
LIN {X 0,Y 62.568,Z 411.056,A -85,B 0,C 180,E1 -29907.804,E2 -29907.804} C_VEL
LIN {X 0,Y 58.99,Z 419.45,A -85,B 0,C 180,E1 -29910.263,E2 -29910.263} C_VEL
LIN {X 0,Y 54.725,Z 427.481,A -85,B 0,C 180,E1 -29913.412,E2 -29913.412} C_VEL
LIN {X 0,Y 50.192,Z 435.227,A -85,B 0,C 180,E1 -29918.038,E2 -29918.038} C_VEL
LIN {X 0,Y 44.771,Z 443.291,A -85,B 0,C 180,E1 -29925.059,E2 -29925.059} C_VEL
LIN {X 0,Y 39.831,Z 450.363,A -85,B 0,C 180,E1 -29935.01,E2 -29935.01} C_VEL
LIN {X 0,Y 36.333,Z 455.937,A -85,B 0,C 180,E1 -29947.241,E2 -29947.241} C_VEL
LIN {X 0,Y 34.487,Z 461.084,A -85,B 0,C 180,E1 -29964.152,E2 -29964.152} C_VEL
LIN {X 0,Y 34.463,Z 462.539,A -85,B 0,C 180,E1 -29970,E2 -29970} C_VEL
LIN {X 0,Y 34.825,Z 464.749,A -85,B 0,C 180,E1 -29981.642,E2 -29981.642} C_VEL
LIN {X 0,Y 36.315,Z 466.404,A -85,B 0,C 180,E1 -29992.771,E2 -29992.771} C_VEL
LIN {X 0,Y 39.032,Z 467.61,A -85,B 0,C 180,E1 -30002.694,E2 -30002.694} C_VEL
LIN {X 0,Y 42.769,Z 468.39,A -85,B 0,C 180,E1 -30011.092,E2 -30011.092} C_VEL
LIN {X 0,Y 47.231,Z 468.637,A -85,B 0,C 180,E1 -30018.071,E2 -30018.071} C_VEL
LIN {X 0,Y 52.352,Z 468.387,A -85,B 0,C 180,E1 -30023.653,E2 -30023.653} C_VEL
LIN {X 0,Y 57.917,Z 467.723,A -85,B 0,C 180,E1 -30028.145,E2 -30028.145} C_VEL
LIN {X 0,Y 63.828,Z 466.627,A -85,B 0,C 180,E1 -30031.744,E2 -30031.744} C_VEL
LIN {X 0,Y 73.066,Z 463.944,A -85,B 0,C 180,E1 -30036.028,E2 -30036.028} C_VEL
LIN {X 0,Y 79.408,Z 461.581,A -85,B 0,C 180,E1 -30038.321,E2 -30038.321} C_VEL
LIN {X 0,Y 85.911,Z 458.571,A -85,B 0,C 180,E1 -30040.175,E2 -30040.175} C_VEL
LIN {X 0,Y 92.435,Z 454.905,A -85,B 0,C 180,E1 -30041.873,E2 -30041.873} C_VEL
LIN {X 0,Y 102.41,Z 448.127,A -85,B 0,C 180,E1 -30043.89,E2 -30043.89} C_VEL
LIN {X 0,Y 110.851,Z 440.793,A -85,B 0,C 180,E1 -30045.2,E2 -30045.2} C_VEL
LIN {X 0,Y 117.815,Z 433.415,A -85,B 0,C 180,E1 -30046.124,E2 -30046.124} C_VEL
LIN {X 0,Y 120.627,Z 430.101,A -85,B 0,C 180,E1 -30046.524,E2 -30046.524} C_VEL
